// TIA Portal V17 program export: 3 tag tables, 14 data types, 19 data blocks, 63 code blocks (in call order from the OBs), 4 instance data blocks

VAR_GLOBAL   // PLC tag table "Default tag table"
   System_Byte AT %MB0 : Byte;
   FirstScan AT %M0.0 : Bool;
   DiagStatusUpdate AT %M0.1 : Bool;
   AlwaysTRUE AT %M0.2 : Bool;
   AlwaysFALSE AT %M0.3 : Bool;
   Clock_Byte AT %MB1 : Byte;
   Clock_10Hz AT %M1.0 : Bool;
   Clock_5Hz AT %M1.1 : Bool;
   "Clock_2.5Hz" AT %M1.2 : Bool;
   Clock_2Hz AT %M1.3 : Bool;
   "Clock_1.25Hz" AT %M1.4 : Bool;
   Clock_1Hz AT %M1.5 : Bool;
   "Clock_0.625Hz" AT %M1.6 : Bool;
   "Clock_0.5Hz" AT %M1.7 : Bool;
END_VAR

VAR_GLOBAL   // PLC tag table "CPG_Constants"
END_VAR
VAR_GLOBAL CONSTANT   // user constants
   CPG_NO_OF_ELEMENTS_EVENT_STATUS_UPPER_LIM : Int := 29;   // Number of Alarms, Warning and PackML Status events used by Event Status UDT (Array size of 0..x)
   CPG_NO_OF_ADMIN_EVENTS_UPPER_LIM : Int := 9;   // Number of Alarms and Warning events found in the PackTags Admin Area - active alarms / warnings. (Array size of 0..x)
   CPG_NO_OF_ADMIN_EVENTS_HISTORY_UPPER_LIM : Int := 9;   // Number of Alarms and Warning events found in the PackTags Admin Area - historical alarms / warnings. (Array size of 0..x)
   CPG_NO_OF_PROD_CONSUMED_COUNT_UPPER_LIM : Int := 0;   // Number of Prod Consumed Counter Array Size (PackTags Admin) (Array size of 0..x)
   CPG_NO_OF_PROD_PROCESSED_COUNT_UPPER_LIM : Int := 0;   // Number of Prod Processed Counter Array Size (PackTags Admin) (Array size of 0..x)
   CPG_NO_OF_PROD_DEFECTIVE_COUNT_UPPER_LIM : Int := 0;   // Number of Prod Defective Counter Array Size (PackTags Admin) (Array size of 0..x)
   CPG_NO_OF_STS_ELEMENTS_EVENT_SUM_UPPER_LIM : Int := 99;   // Number of Alarms, Warning and PackML Status events used by Event Summation UDT (Array size of 0..x)
   CPG_NO_OF_HMI_SORT_EVENTS_UPPER_LIM : Int := 19;   // Number of Alarms and Warning events found for the HMI area - sorted HMI alarms / warnings. (Array size of 0..x)
   CPG_NO_OF_CFG_ALARMS_UPPER_LIM : Int := 39;   // Number of Cfg Alarm event configurations (Array size of 0..x)
   CPG_NO_OF_CFG_WARNINGS_UPPER_LIM : Int := 29;   // Number of Cfg Warning event configurations (Array size of 0..x)
   CPG_NO_OF_CFG_STATUS_UPPER_LIM : Int := 19;   // Number of Cfg Status event configurations (Array size of 0..x)
   CPG_NO_OF_STATUS_PARAMETERS_UPPER_LIM : Int := 0;   // Number of Status Parameters (Array size of 0..x)
   CPG_NO_OF_COMMAND_PARAMETERS_UPPER_LIM : Int := 0;   // Number of Command Parameters (Array size of 0..x)
   CPG_NO_OF_ADMIN_PARAMETERS_UPPER_LIM : Int := 0;   // Number of Admin Parameters (Array size of 0..x)
   CPG_NO_OF_RECIPE_UPPER_LIM : Int := 20;   // Number of Project Recipies (Array size of 0..x)
   CPG_NO_OF_SETPOINT_REAL_UPPER_LIM : Int := 0;   // Number of Setpoints with a REAL type (Array size of 0..x)
   CPG_NO_OF_SETPOINT_DINT_UPPER_LIM : Int := 0;   // Number of Setpoints with a DINT type (Array size of 0..x)
   CPG_NO_OF_SETPOINT_BOOL_UPPER_LIM : Int := 0;   // Number of Setpoints with a BOOL type (Array size of 0..x)
   CPG_NO_OF_SETPOINT_STRING_UPPER_LIM : Int := 0;   // Number of Setpoints with a STRING type (Array size of 0..x)
   CPG_PARTEO_NO_OF_ERRORS_UPPER_LIM : Int := 100;   // Number of Unique Error IDs tracked by PARETO Error Blocks
END_VAR

VAR_GLOBAL   // PLC tag table "LPMLV30_Constants"
END_VAR
VAR_GLOBAL CONSTANT   // user constants
   LPMLV30_MODE_INVALID : DInt := 0;   // OMAC PackMLV30 unit mode Invalid
   LPMLV30_MODE_PRODUCTION : DInt := 1;   // OMAC PackMLV30 unit mode Production
   LPMLV30_MODE_MAINTENANCE : DInt := 2;   // OMAC PackMLV30 unit mode Maintenance
   LPMLV30_MODE_MANUAL : DInt := 3;   // OMAC PackMLV30 unit mode Manual
   LPMLV30_MODE_USER_01 : DInt := 4;   // OMAC PackMLV30 user-defined unit mode 01
   LPMLV30_MODE_USER_02 : DInt := 5;   // OMAC PackMLV30 user-defined unit mode 02
   LPMLV30_MODE_USER_03 : DInt := 6;   // OMAC PackMLV30 user-defined unit mode 03
   LPMLV30_MODE_USER_04 : DInt := 7;   // OMAC PackMLV30 user-defined unit mode 04
   LPMLV30_MODE_USER_05 : DInt := 8;   // OMAC PackMLV30 user-defined unit mode 05
   LPMLV30_MODE_USER_06 : DInt := 9;   // OMAC PackMLV30 user-defined unit mode 06
   LPMLV30_MODE_USER_07 : DInt := 10;   // OMAC PackMLV30 user-defined unit mode 07
   LPMLV30_MODE_USER_08 : DInt := 11;   // OMAC PackMLV30 user-defined unit mode 08
   LPMLV30_MODE_USER_09 : DInt := 12;   // OMAC PackMLV30 user-defined unit mode 09
   LPMLV30_MODE_USER_10 : DInt := 13;   // OMAC PackMLV30 user-defined unit mode 10
   LPMLV30_MODE_USER_11 : DInt := 14;   // OMAC PackMLV30 user-defined unit mode 11
   LPMLV30_MODE_USER_12 : DInt := 15;   // OMAC PackMLV30 user-defined unit mode 12
   LPMLV30_MODE_USER_13 : DInt := 16;   // OMAC PackMLV30 user-defined unit mode 13
   LPMLV30_MODE_USER_14 : DInt := 17;   // OMAC PackMLV30 user-defined unit mode 14
   LPMLV30_MODE_USER_15 : DInt := 18;   // OMAC PackMLV30 user-defined unit mode 15
   LPMLV30_MODE_USER_16 : DInt := 19;   // OMAC PackMLV30 user-defined unit mode 16
   LPMLV30_MODE_USER_17 : DInt := 20;   // OMAC PackMLV30 user-defined unit mode 17
   LPMLV30_MODE_USER_18 : DInt := 21;   // OMAC PackMLV30 user-defined unit mode 18
   LPMLV30_MODE_USER_19 : DInt := 22;   // OMAC PackMLV30 user-defined unit mode 19
   LPMLV30_MODE_USER_20 : DInt := 23;   // OMAC PackMLV30 user-defined unit mode 20
   LPMLV30_MODE_USER_21 : DInt := 24;   // OMAC PackMLV30 user-defined unit mode 21
   LPMLV30_MODE_USER_22 : DInt := 25;   // OMAC PackMLV30 user-defined unit mode 22
   LPMLV30_MODE_USER_23 : DInt := 26;   // OMAC PackMLV30 user-defined unit mode 23
   LPMLV30_MODE_USER_24 : DInt := 27;   // OMAC PackMLV30 user-defined unit mode 24
   LPMLV30_MODE_USER_25 : DInt := 28;   // OMAC PackMLV30 user-defined unit mode 25
   LPMLV30_MODE_USER_26 : DInt := 29;   // OMAC PackMLV30 user-defined unit mode 26
   LPMLV30_MODE_USER_27 : DInt := 30;   // OMAC PackMLV30 user-defined unit mode 27
   LPMLV30_MODE_USER_28 : DInt := 31;   // OMAC PackMLV30 user-defined unit mode 28
   LPMLV30_STATE_UNDEFINED : DInt := 0;   // OMAC PackMLV30 state Undefined
   LPMLV30_STATE_CLEARING : DInt := 1;   // OMAC PackMLV30 state Clearing
   LPMLV30_STATE_STOPPED : DInt := 2;   // OMAC PackMLV30 state Stopped
   LPMLV30_STATE_STARTING : DInt := 3;   // OMAC PackMLV30 state Starting
   LPMLV30_STATE_IDLE : DInt := 4;   // OMAC PackMLV30 state Idle
   LPMLV30_STATE_SUSPENDED : DInt := 5;   // OMAC PackMLV30 state Suspended
   LPMLV30_STATE_EXECUTE : DInt := 6;   // OMAC PackMLV30 state Execute
   LPMLV30_STATE_STOPPING : DInt := 7;   // OMAC PackMLV30 state Stopping
   LPMLV30_STATE_ABORTING : DInt := 8;   // OMAC PackMLV30 state Aborting
   LPMLV30_STATE_ABORTED : DInt := 9;   // OMAC PackMLV30 state Aborted
   LPMLV30_STATE_HOLDING : DInt := 10;   // OMAC PackMLV30 state Holding
   LPMLV30_STATE_HELD : DInt := 11;   // OMAC PackMLV30 state Held
   LPMLV30_STATE_UNHOLDING : DInt := 12;   // OMAC PackMLV30 state Unholding
   LPMLV30_STATE_SUSPENDING : DInt := 13;   // OMAC PackMLV30 state Suspending
   LPMLV30_STATE_UNSUSPENDING : DInt := 14;   // OMAC PackMLV30 state Unsuspending
   LPMLV30_STATE_RESETTING : DInt := 15;   // OMAC PackMLV30 state Resetting
   LPMLV30_STATE_COMPLETING : DInt := 16;   // OMAC PackMLV30 state Completing
   LPMLV30_STATE_COMPLETE : DInt := 17;   // OMAC PackMLV30 state Complete
   LPMLV30_CMD_UNDEFINED : DInt := 0;   // OMAC PackMLV30 control command Undefined
   LPMLV30_CMD_RESET : DInt := 1;   // OMAC PackMLV30 control command Reset
   LPMLV30_CMD_START : DInt := 2;   // OMAC PackMLV30 control command Start
   LPMLV30_CMD_STOP : DInt := 3;   // OMAC PackMLV30 control command Stop
   LPMLV30_CMD_HOLD : DInt := 4;   // OMAC PackMLV30 control command Hold
   LPMLV30_CMD_UNHOLD : DInt := 5;   // OMAC PackMLV30 control command Unhold
   LPMLV30_CMD_SUSPEND : DInt := 6;   // OMAC PackMLV30 control command Suspend
   LPMLV30_CMD_UNSUSPEND : DInt := 7;   // OMAC PackMLV30 control command Unsuspend
   LPMLV30_CMD_ABORT : DInt := 8;   // OMAC PackMLV30 control command Abort
   LPMLV30_CMD_CLEAR : DInt := 9;   // OMAC PackMLV30 control command Clear
   LPMLV30_CMD_COMPLETE : DInt := 10;   // OMAC PackMLV30 control command Complete
   LPMLV30_LANGUAGE_1 : Int := 0;   // Texts in 1st language (default English)
   LPMLV30_LANGUAGE_2 : Int := 1;   // Texts in 2nd language (default German)
   LPMLV30_DIAG_BUFFER_UPPER_LIM : Int := 15;   // Diagnostics buffer array upper boundary (0-based)
   LPMLV30_LANGUAGES_UPPER_LIM : Int := 2;   // (Number of languages - 1) -> Array[0..LPMLV30_LANGUAGES_UPPER_LIM]
   LPMLV30_MODES_UPPER_LIM : Int := 4;   // (Number of unit modes - 1) -> Array[0..LPMLV30_MODES_UPPER_LIM]
   LPMLV30_STATES_UPPER_LIM : Int := 17;   // (Number of states - 1) -> Array[0..LPMLV30_STATES_UPPER_LIM] (SHOULD ALWAYS BE 17!)
   LPMLV30_MAX_MODES_UPPER_LIM : Int := 31;   // (Maximum number of unit modes - 1) -> Array[0..LPMLV30_MAX_MODES_UPPER_LIM]
END_VAR

TYPE "CPG_typeEventCfg"
// stored: IsFailsafeCompliant false
   STRUCT
      ID : Int;   // ID Value - from PackTags Reason Code, 1=E-Stop pushed, 3=Main off, etc.
      value : Int;   // Reason Code 'Value' - allows for detailed breakdown of ID, ie 1=Discharge,
      message : Array[0.."LPMLV30_LANGUAGES_UPPER_LIM"] of String[60];   // Alarm Message - 0=English, 1=German, 2=Spanish, 3=Italian, 4=French
      category : Int;   // Category Value (0-9)
   END_STRUCT;
END_TYPE

TYPE "CPG_typeEventStatus"
// stored: IsFailsafeCompliant false
   STRUCT
      sts_FirstOutEvent { S7_SetPoint := 'True'} : "CPG_typeEvent";   // Event Info of the very first active event (irregardeless of the cat)
      sts_FirstOutEventCat { S7_SetPoint := 'True'} : Array[0..9] of "CPG_typeEvent";
      sts_Events { S7_SetPoint := 'True'} : Array[0.."CPG_NO_OF_ELEMENTS_EVENT_STATUS_UPPER_LIM"] of "CPG_typeEvent";
      sts_NumEvents : Int;   // Number of all current active events
      sts_NumAllEvents : Int;   // Number of all current events
      out_ZeroEvent { S7_SetPoint := 'True'} : "CPG_typeEvent";   // null event information
      sts_Category_0_Latched : Bool;   // Category 0 Event - latched (require reset cmd)
      sts_Category_1_Latched : Bool;   // Category 1 Event - latched (require reset cmd)
      sts_Category_2_Latched : Bool;   // Category 2 Event - latched (require reset cmd)
      sts_Category_3_Latched : Bool;   // Category 3 Event - latched (require reset cmd)
      sts_Category_4_Latched : Bool;   // Category 4 Event - latched (require reset cmd)
      sts_Category_5_Latched : Bool;   // Category 5 Event - latched (require reset cmd)
      sts_Category_6_Latched : Bool;   // Category 6 Event - latched (require reset cmd)
      sts_Category_7_Latched : Bool;   // Category 7 Event - latched (require reset cmd)
      sts_Category_8_Latched : Bool;   // Category 8 Event - latched (require reset cmd)
      sts_Category_9_Latched : Bool;   // Category 9 Event - latched (require reset cmd)
      sts_Category_0_NotLatched : Bool;   // Category 0 Event - NotLatched (currently active)
      sts_Category_1_NotLatched : Bool;   // Category 1 Event - NotLatched (currently active)
      sts_Category_2_NotLatched : Bool;   // Category 2 Event - NotLatched (currently active)
      sts_Category_3_NotLatched : Bool;   // Category 3 Event - NotLatched (currently active)
      sts_Category_4_NotLatched : Bool;   // Category 4 Event - NotLatched (currently active)
      sts_Category_5_NotLatched : Bool;   // Category 5 Event - NotLatched (currently active)
      sts_Category_6_NotLatched : Bool;   // Category 6 Event - NotLatched (currently active)
      sts_Category_7_NotLatched : Bool;   // Category 7 Event - NotLatched (currently active)
      sts_Category_8_NotLatched : Bool;   // Category 8 Event - NotLatched (currently active)
      sts_Category_9_NotLatched : Bool;   // Category 9 Event - NotLatched (currently active)
      sts_CurrentActiveEvent : Bool;   // Active # of Event
      wrk_ResetID : Int;   // Working Variable - DO NOT MODIFY
      wrk_EventArraySize : Int;   // Working Variable - DO NOT MODIFY
      wrk_UpdateEventListID : Int;   // Working Variable - DO NOT MODIFY
      wrk_LanguageSelection : Int;   // This is the value of language selected in the HMI
      wrk_MessagePrefix : String[10];   // Working Variable - DO NOT MODIFY
   END_STRUCT;
END_TYPE

TYPE "CPG_typeEventSummation"
// stored: IsFailsafeCompliant false
   STRUCT
      sts_FirstOutEvent { S7_SetPoint := 'True'} : "CPG_typeEvent";   // First Out (Stop Reason) Event
      sts_FirstOutEventCat { S7_SetPoint := 'True'} : Array[0..9] of "CPG_typeEvent";   // First Out (Stop Reason) Event by Category\
      sts_Events { S7_SetPoint := 'True'} : Array[0.."CPG_NO_OF_STS_ELEMENTS_EVENT_SUM_UPPER_LIM"] of "CPG_typeEvent";   // All Active Events
      sts_NumEvents : Int;   // Number of Active Events
      sts_Category_0_Latched : Bool;   // Category 0 Event - latched (require reset cmd)
      sts_Category_1_Latched : Bool;   // Category 1 Event - latched (require reset cmd)
      sts_Category_2_Latched : Bool;   // Category 2 Event - latched (require reset cmd)
      sts_Category_3_Latched : Bool;   // Category 3 Event - latched (require reset cmd)
      sts_Category_4_Latched : Bool;   // Category 4 Event - latched (require reset cmd)
      sts_Category_5_Latched : Bool;   // Category 5 Event - latched (require reset cmd)
      sts_Category_6_Latched : Bool;   // Category 6 Event - latched (require reset cmd)
      sts_Category_7_Latched : Bool;   // Category 7 Event - latched (require reset cmd)
      sts_Category_8_Latched : Bool;   // Category 8 Event - latched (require reset cmd)
      sts_Category_9_Latched : Bool;   // Category 9 Event - latched (require reset cmd)
      sts_Category_0_NotLatched : Bool;   // Category 0 Event - NotLatched (currently active)
      sts_Category_1_NotLatched : Bool;   // Category 1 Event - NotLatched (currently active)
      sts_Category_2_NotLatched : Bool;   // Category 2 Event - NotLatched (currently active)
      sts_Category_3_NotLatched : Bool;   // Category 3 Event - NotLatched (currently active)
      sts_Category_4_NotLatched : Bool;   // Category 4 Event - NotLatched (currently active)
      sts_Category_5_NotLatched : Bool;   // Category 5 Event - NotLatched (currently active)
      sts_Category_6_NotLatched : Bool;   // Category 6 Event - NotLatched (currently active)
      sts_Category_7_NotLatched : Bool;   // Category 7 Event - NotLatched (currently active)
      sts_Category_8_NotLatched : Bool;   // Category 8 Event - NotLatched (currently active)
      sts_Category_9_NotLatched : Bool;   // Category 9 Event - NotLatched (currently active)
      sts_CurrentActiveEvent : Bool;   // Event Active = 1, not active = 0
      wrk_EventArraySize : Int;   // Maximum Array Size - DO NOT MODIFY
      wrk_Category_0_Latched : Bool;   // Working Variable - DO NOT MODIFY
      wrk_Category_1_Latched : Bool;   // Working Variable - DO NOT MODIFY
      wrk_Category_2_Latched : Bool;   // Working Variable - DO NOT MODIFY
      wrk_Category_3_Latched : Bool;   // Working Variable - DO NOT MODIFY
      wrk_Category_4_Latched : Bool;   // Working Variable - DO NOT MODIFY
      wrk_Category_5_Latched : Bool;   // Working Variable - DO NOT MODIFY
      wrk_Category_6_Latched : Bool;   // Working Variable - DO NOT MODIFY
      wrk_Category_7_Latched : Bool;   // Working Variable - DO NOT MODIFY
      wrk_Category_8_Latched : Bool;   // Working Variable - DO NOT MODIFY
      wrk_Category_9_Latched : Bool;   // Working Variable - DO NOT MODIFY
      wrk_Category_0_NotLatched : Bool;   // Working Variable - DO NOT MODIFY
      wrk_Category_1_NotLatched : Bool;   // Working Variable - DO NOT MODIFY
      wrk_Category_2_NotLatched : Bool;   // Working Variable - DO NOT MODIFY
      wrk_Category_3_NotLatched : Bool;   // Working Variable - DO NOT MODIFY
      wrk_Category_4_NotLatched : Bool;   // Working Variable - DO NOT MODIFY
      wrk_Category_5_NotLatched : Bool;   // Working Variable - DO NOT MODIFY
      wrk_Category_6_NotLatched : Bool;   // Working Variable - DO NOT MODIFY
      wrk_Category_7_NotLatched : Bool;   // Working Variable - DO NOT MODIFY
      wrk_Category_8_NotLatched : Bool;   // Working Variable - DO NOT MODIFY
      wrk_Category_9_NotLatched : Bool;   // Working Variable - DO NOT MODIFY
      wrk_CurrentActiveEvent : Bool;   // Working Variable - DO NOT MODIFY
   END_STRUCT;
END_TYPE

TYPE "CPG_typeMessagePrefix"
// stored: IsFailsafeCompliant false
   STRUCT
      messagePrefix : Array[0.."LPMLV30_LANGUAGES_UPPER_LIM"] of String[30];   // Multi-Lingual Message for Prefix (i.e 0=EN, 1=DE, 2=SP/ES, 3=IT, 4=FR)
   END_STRUCT;
END_TYPE

TYPE "CPG_typePackML_ModuleSts"
// stored: IsFailsafeCompliant false
   STRUCT
      cmd_Reset : Bool;   // Reset
      sts_Resetting_SC : Bool;   // Resetting State Complete
      cmd_Start : Bool;   // Start
      sts_Starting_SC : Bool;   // Starting State Complete
      cmd_Stop : Bool;   // Stop
      sts_Stopping_SC : Bool;   // Stopping State Complete
      cmd_Hold : Bool;   // Hold
      sts_Holding_SC : Bool;   // Holding State Complete
      cmd_UnHold : Bool;   // UnHold
      sts_UnHolding_SC : Bool;   // UnHolding State Complete
      cmd_Suspend : Bool;   // Suspend
      sts_Suspending_SC : Bool;   // Suspending State Complete
      cmd_UnSuspend : Bool;   // UnSuspend
      sts_UnSuspending_SC : Bool;   // UnSuspending State Complete
      cmd_Abort : Bool;   // Abort
      sts_Aborting_SC : Bool;   // Aborting State Complete
      cmd_Clear : Bool;   // Clear
      sts_Clearing_SC : Bool;   // Clearing State Complete
      sts_Execute_SC : Bool;   // Execute State Complete
      sts_Completing_SC : Bool;   // Completing State Complete
      moduleActive : Bool;   // Module Active Bit
      ONS : Bool;   // Internal One Shot Bit - Do not modify
   END_STRUCT;
END_TYPE

TYPE "CPG_typeParameter(DINT)"
// stored: IsFailsafeCompliant false
   STRUCT
      ID : DInt;   // Parameter ID - This is the arbitrary (user defined) ID value of the parameter
      "Name" : String[24];   // Parameter Name - The literal parameter name is used to describe the parameter number and its associated value (e.g. Glue Temp)
      Unit : String[5];   // Parameter Unit of Measure - The parameter unit is used to describe the unit of measure of the parameter and its associated value (e.g. DegF)
      Value : DInt;   // Parameter Value - This is the numeric or string value of the parameter (e.g. 100)
   END_STRUCT;
END_TYPE

TYPE "CPG_typeParameter(Real)"
// stored: IsFailsafeCompliant false
   STRUCT
      ID : DInt;   // Parameter ID - This is the arbitrary (user defined) ID value of the parameter
      "Name" : String[24];   // Parameter Name - The literal parameter name is used to describe the parameter number and its associated value (e.g. Glue Temp)
      Unit : String[5];   // Parameter Unit of Measure - The parameter unit is used to describe the unit of measure of the parameter and its associated value (e.g. DegF)
      Value : Real;   // Parameter Value - This is the numeric or string value of the parameter (e.g. 100.2)
   END_STRUCT;
END_TYPE

TYPE "CPG_typeParameter(String)"
// stored: IsFailsafeCompliant false
   STRUCT
      ID : DInt;   // Parameter ID - This is the arbitrary (user defined) ID value of the parameter
      "Name" : String[24];   // Parameter Name - The literal parameter name is used to describe the parameter number and its associated value (e.g. Glue Temp)
      Unit : String[5];   // Parameter Unit of Measure - The parameter unit is used to describe the unit of measure of the parameter and its associated value (e.g. DegF)
      Value : String[24];   // Parameter Value - This is the numeric or string value of the parameter (e.g. '6ES7518-4AP00-0AB0')
   END_STRUCT;
END_TYPE

TYPE "CPG_typeProdCount(DINT)"
// stored: IsFailsafeCompliant false
   STRUCT
      ID : DInt;   // Product ID - This is the arbitrary (user defined) ID value of the consumed production material
      "Name" : String[24];   // Descriptive name - The name is used to literally describe the material ID, and its associated material
      Unit : String[5];   // Unit of measure - The unit tag is used to describe the names associated with a specific material used by the machine
      Count : DInt;   // Value - The count value is used as a variable for displaying information about the amount of consumed
      AccCount : DInt;   // Value - The accumulative count value is used as a variable for displaying information about the total amount of consumed production material
   END_STRUCT;
END_TYPE

TYPE "CPG_typeSortFilter"
// stored: IsFailsafeCompliant false
   STRUCT
      cmdFilterActiveEvents : Bool;   // Filter for Active events: 1=only show active events; 0=show all events
      cmdFilterCategory : Bool;   // Filter by Category: filter events to show only selected category number
      cmdSortCategory : Bool;   // Sort by Category: 1=sort events by ascending category number
      cfgTimeSortDirection : Bool;   // Sort by Time: 1=newest first; 0=oldest first
      cfgEventListOffset : Int;   // Commanded event list offset (used for scrolling)
      cfgFilterCategory : Int;   // Filter by Category: filtered category number
   END_STRUCT;
END_TYPE

TYPE "typeLPMLV30_Configuration"
TITLE = typeLPMLV30_Configuration
// Support: tech.team.motioncontrol@siemens.com 
// Fax: +49 (0) 9131/98-1297
// stored: IsFailsafeCompliant false
   STRUCT
      disabledUnitModes : Array[0.."LPMLV30_MAX_MODES_UPPER_LIM"] of Bool;   // TRUE: Disable unit mode xx
      disabledStatesInUnitModes : Array[0.."LPMLV30_MAX_MODES_UPPER_LIM"] of DInt;   // TRUE: Disable states in unit mode (bit number = state number)
   END_STRUCT;
   // disabledUnitModes[0..11] := false;
   // disabledUnitModes[12..31] := true;
   // disabledStatesInUnitModes[0..31] := 0;
END_TYPE

TYPE "typeLPMLV30_Diagnostics"
TITLE = typeLPMLV30_Diagnostics
// Support: tech.team.motioncontrol@siemens.com 
// Fax: +49 (0) 9131/98-1297
// stored: IsFailsafeCompliant false
   STRUCT
      bufferIndex : Int := -1;   // Index of actual buffer entry
      buffer { S7_SetPoint := 'True'} : Array[0.."LPMLV30_DIAG_BUFFER_UPPER_LIM"] of "typeLPMLV30_DiagnosticsEntry";   // Diagnostics information buffer
   END_STRUCT;
END_TYPE

TYPE "typeLPMLV30_DiagnosticsEntry"
TITLE = typeLPMLV30_DiagnosticsEntry
// Support: tech.team.motioncontrol@siemens.com 
// Fax: +49 (0) 9131/98-1297
// stored: IsFailsafeCompliant false
   STRUCT
      timestamp : DTL := DTL#1970-01-01-00:00:00;   // Timestamp for this entry
      UnitModeCurrent : Byte := 16#00;   // Current unit mode
      StateCurrent : Byte := 16#00;   // Current state
      UnitMode : Byte := 16#00;   // Requested unit mode
      CntrlCmd : Byte := 16#00;   // Request control command
      SC : Bool := false;   // State complete signal
      message : Byte := 16#00;   // Message for this entry
   END_STRUCT;
END_TYPE

TYPE "typeLPMLV30_NamesConfiguration"
TITLE = typeLPMLV30_NamesConfiguration
// Support: tech.team.motioncontrol@siemens.com 
// Fax: +49 (0) 9131/98-1297
// stored: IsFailsafeCompliant false
   STRUCT
      unitModesNames : Array[0.."LPMLV30_LANGUAGES_UPPER_LIM", 0.."LPMLV30_MODES_UPPER_LIM"] of String[18];   // Names of unit modes [First index language, Second unit mode no]
      statesNames : Array[0.."LPMLV30_LANGUAGES_UPPER_LIM", 0.."LPMLV30_STATES_UPPER_LIM"] of String[16];   // Names of states [First index language, Second state no]
   END_STRUCT;
   // unitModesNames[0,0] := 'Invalid';
   // unitModesNames[0,1] := 'Production';
   // unitModesNames[0,2] := 'Maintenance';
   // unitModesNames[0,3] := 'Manual';
   // unitModesNames[0,4] := 'User Mode 01';
   // unitModesNames[1,0] := 'Undefiniert';
   // unitModesNames[1,1] := 'Produktion';
   // unitModesNames[1,2] := 'Wartung';
   // unitModesNames[1,3] := 'Hand';
   // unitModesNames[1,4] := 'Benutzer Mode 01';
   // statesNames[0,0] := 'Undefined';
   // statesNames[0,1] := 'Clearing';
   // statesNames[0,2] := 'Stopped';
   // statesNames[0,3] := 'Starting';
   // statesNames[0,4] := 'Idle';
   // statesNames[0,5] := 'Suspended';
   // statesNames[0,6] := 'Execute';
   // statesNames[0,7] := 'Stopping';
   // statesNames[0,8] := 'Aborting';
   // statesNames[0,9] := 'Aborted';
   // statesNames[0,10] := 'Holding';
   // statesNames[0,11] := 'Held';
   // statesNames[0,12] := 'UnHolding';
   // statesNames[0,13] := 'Suspending';
   // statesNames[0,14] := 'UnSuspending';
   // statesNames[0,15] := 'Resetting';
   // statesNames[0,16] := 'Completing';
   // statesNames[0,17] := 'Complete';
   // statesNames[1,0] := 'Undefiniert';
   // statesNames[1,1] := 'Clearing';
   // statesNames[1,2] := 'Stopped';
   // statesNames[1,3] := 'Starting';
   // statesNames[1,4] := 'Idle';
   // statesNames[1,5] := 'Suspended';
   // statesNames[1,6] := 'Execute';
   // statesNames[1,7] := 'Stopping';
   // statesNames[1,8] := 'Aborting';
   // statesNames[1,9] := 'Aborted';
   // statesNames[1,10] := 'Holding';
   // statesNames[1,11] := 'Held';
   // statesNames[1,12] := 'UnHolding';
   // statesNames[1,13] := 'Suspending';
   // statesNames[1,14] := 'UnSuspending';
   // statesNames[1,15] := 'Resetting';
   // statesNames[1,16] := 'Completing';
   // statesNames[1,17] := 'Complete';
END_TYPE

DATA_BLOCK "EM00"   // DB31649
TITLE = EM00
{ S7_Optimized_Access := 'TRUE' }
AUTHOR : tech.team.motioncontrol@siemens.com
FAMILY : CPG
VERSION : 1.1
// Support: tech.team.motioncontrol@siemens.com
// stored: AutoNumber true, DBAccessibleFromOPCUA true, DBAccessibleFromWebserver true, IsOnlyStoredInLoadMemory false, IsRetainMemResEnabled false, IsWriteProtectedInAS false, MemoryReserve 100
   VAR
      PackML_Sts { ExternalWritable := 'False'} : Struct   // PackML Module Status - EM and all control modules
         Unit { ExternalWritable := 'False'; S7_SetPoint := 'True'} : "CPG_typePackML_ModuleSts";   // PackML Module Status - EM - master status
         Alarm { ExternalWritable := 'False'; S7_SetPoint := 'True'} : "CPG_typePackML_ModuleSts";   // PackML Module Status - alarm status
         CM01 { ExternalWritable := 'False'; S7_SetPoint := 'True'} : "CPG_typePackML_ModuleSts";   // PackML Module Status - CM 01
         CM02 { ExternalWritable := 'False'; S7_SetPoint := 'True'} : "CPG_typePackML_ModuleSts";   // PackML Module Status - CM 02
         CM03 { ExternalWritable := 'False'; S7_SetPoint := 'True'} : "CPG_typePackML_ModuleSts";   // PackML Module Status - CM 03
         CM04 { ExternalWritable := 'False'; S7_SetPoint := 'True'} : "CPG_typePackML_ModuleSts";   // PackML Module Status - CM 04
         CM05 { ExternalWritable := 'False'; S7_SetPoint := 'True'} : "CPG_typePackML_ModuleSts";   // PackML Module Status - CM 05
         CM06 { ExternalWritable := 'False'; S7_SetPoint := 'True'} : "CPG_typePackML_ModuleSts";   // PackML Module Status - CM 06
         CM07 { ExternalWritable := 'False'; S7_SetPoint := 'True'} : "CPG_typePackML_ModuleSts";   // PackML Module Status - CM 07
         CM08 { ExternalWritable := 'False'; S7_SetPoint := 'True'} : "CPG_typePackML_ModuleSts";   // PackML Module Status - CM 08
         CM09 { ExternalWritable := 'False'; S7_SetPoint := 'True'} : "CPG_typePackML_ModuleSts";   // PackML Module Status - CM 09
         CM10 { ExternalWritable := 'False'; S7_SetPoint := 'True'} : "CPG_typePackML_ModuleSts";   // PackML Module Status - CM 10
      END_STRUCT;
      Alarm { ExternalAccessible := 'False'; ExternalVisible := 'False'; ExternalWritable := 'False'; S7_SetPoint := 'True'} : "CPG_typeEventStatus";   // Alarm Event Status - EM00 Status
      Warning { ExternalAccessible := 'False'; ExternalVisible := 'False'; ExternalWritable := 'False'; S7_SetPoint := 'True'} : "CPG_typeEventStatus";   // Warning Event Status - EM00 Status
      Status { ExternalAccessible := 'False'; ExternalVisible := 'False'; ExternalWritable := 'False'; S7_SetPoint := 'True'} : "CPG_typeEventStatus";   // Event Status - EM00 Status
   END_VAR
BEGIN
END_DATA_BLOCK

DATA_BLOCK "EM01"   // DB31669
TITLE = EM01
{ S7_Optimized_Access := 'TRUE' }
AUTHOR : tech.team.motioncontrol@siemens.com
FAMILY : CPG
VERSION : 1.0
// Support: tech.team.motioncontrol@siemens.com
// Fax: +49 (0) 9131/98-1297
// stored: AutoNumber true, DBAccessibleFromOPCUA true, DBAccessibleFromWebserver true, IsOnlyStoredInLoadMemory false, IsRetainMemResEnabled false, IsWriteProtectedInAS false, MemoryReserve 100
   VAR
      PackML_Sts { ExternalWritable := 'False'} : Struct   // PackML Module Status - EM and all control modules
         Unit { ExternalWritable := 'False'; S7_SetPoint := 'True'} : "CPG_typePackML_ModuleSts";   // PackML Module Status - EM - master status
         Alarm { ExternalWritable := 'False'; S7_SetPoint := 'True'} : "CPG_typePackML_ModuleSts";   // PackML Module Status - alarm status
         CM01 { ExternalWritable := 'False'; S7_SetPoint := 'True'} : "CPG_typePackML_ModuleSts";   // PackML Module Status - CM 01
         CM02 { ExternalWritable := 'False'; S7_SetPoint := 'True'} : "CPG_typePackML_ModuleSts";   // PackML Module Status - CM 02
         CM03 { ExternalWritable := 'False'; S7_SetPoint := 'True'} : "CPG_typePackML_ModuleSts";   // PackML Module Status - CM 03
         CM04 { ExternalWritable := 'False'; S7_SetPoint := 'True'} : "CPG_typePackML_ModuleSts";   // PackML Module Status - CM 04
         CM05 { ExternalWritable := 'False'; S7_SetPoint := 'True'} : "CPG_typePackML_ModuleSts";   // PackML Module Status - CM 05
         CM06 { ExternalWritable := 'False'; S7_SetPoint := 'True'} : "CPG_typePackML_ModuleSts";   // PackML Module Status - CM 06
         CM07 { ExternalWritable := 'False'; S7_SetPoint := 'True'} : "CPG_typePackML_ModuleSts";   // PackML Module Status - CM 07
         CM08 { ExternalWritable := 'False'; S7_SetPoint := 'True'} : "CPG_typePackML_ModuleSts";   // PackML Module Status - CM 08
         CM09 { ExternalWritable := 'False'; S7_SetPoint := 'True'} : "CPG_typePackML_ModuleSts";   // PackML Module Status - CM 09
         CM10 { ExternalWritable := 'False'; S7_SetPoint := 'True'} : "CPG_typePackML_ModuleSts";   // PackML Module Status - CM 10
      END_STRUCT;
      Alarm { ExternalAccessible := 'False'; ExternalVisible := 'False'; ExternalWritable := 'False'; S7_SetPoint := 'True'} : "CPG_typeEventStatus";   // Alarm Event Status - EM01 Status
      Warning { ExternalAccessible := 'False'; ExternalVisible := 'False'; ExternalWritable := 'False'; S7_SetPoint := 'True'} : "CPG_typeEventStatus";   // Warning Event Status - EM01 Status
      Status { ExternalAccessible := 'False'; ExternalVisible := 'False'; ExternalWritable := 'False'; S7_SetPoint := 'True'} : "CPG_typeEventStatus";   // Event Status - EM01 Status
   END_VAR
BEGIN
END_DATA_BLOCK

DATA_BLOCK "EM02"   // DB31689
TITLE = EM02
{ S7_Optimized_Access := 'TRUE' }
AUTHOR : tech.team.motioncontrol@siemens.com
FAMILY : CPG
VERSION : 1.0
// Support: tech.team.motioncontrol@siemens.com
// Fax: +49 (0) 9131/98-1297
// stored: AutoNumber true, DBAccessibleFromOPCUA true, DBAccessibleFromWebserver true, IsOnlyStoredInLoadMemory false, IsRetainMemResEnabled false, IsWriteProtectedInAS false, MemoryReserve 100
   VAR
      PackML_Sts { ExternalWritable := 'False'} : Struct   // PackML Module Status - EM and all control modules
         Unit { ExternalWritable := 'False'; S7_SetPoint := 'True'} : "CPG_typePackML_ModuleSts";   // PackML Module Status - EM - master status
         Alarm { ExternalWritable := 'False'; S7_SetPoint := 'True'} : "CPG_typePackML_ModuleSts";   // PackML Module Status - alarm status
         CM01 { ExternalWritable := 'False'; S7_SetPoint := 'True'} : "CPG_typePackML_ModuleSts";   // PackML Module Status - CM 01
         CM02 { ExternalWritable := 'False'; S7_SetPoint := 'True'} : "CPG_typePackML_ModuleSts";   // PackML Module Status - CM 02
         CM03 { ExternalWritable := 'False'; S7_SetPoint := 'True'} : "CPG_typePackML_ModuleSts";   // PackML Module Status - CM 03
         CM04 { ExternalWritable := 'False'; S7_SetPoint := 'True'} : "CPG_typePackML_ModuleSts";   // PackML Module Status - CM 04
         CM05 { ExternalWritable := 'False'; S7_SetPoint := 'True'} : "CPG_typePackML_ModuleSts";   // PackML Module Status - CM 05
         CM06 { ExternalWritable := 'False'; S7_SetPoint := 'True'} : "CPG_typePackML_ModuleSts";   // PackML Module Status - CM 06
         CM07 { ExternalWritable := 'False'; S7_SetPoint := 'True'} : "CPG_typePackML_ModuleSts";   // PackML Module Status - CM 07
         CM08 { ExternalWritable := 'False'; S7_SetPoint := 'True'} : "CPG_typePackML_ModuleSts";   // PackML Module Status - CM 08
         CM09 { ExternalWritable := 'False'; S7_SetPoint := 'True'} : "CPG_typePackML_ModuleSts";   // PackML Module Status - CM 09
         CM10 { ExternalWritable := 'False'; S7_SetPoint := 'True'} : "CPG_typePackML_ModuleSts";   // PackML Module Status - CM 10
      END_STRUCT;
      Alarm { ExternalAccessible := 'False'; ExternalVisible := 'False'; ExternalWritable := 'False'; S7_SetPoint := 'True'} : "CPG_typeEventStatus";   // Alarm Event Status - EM02 Status
      Warning { ExternalAccessible := 'False'; ExternalVisible := 'False'; ExternalWritable := 'False'; S7_SetPoint := 'True'} : "CPG_typeEventStatus";   // Warning Event Status - EM02 Status
      Status { ExternalAccessible := 'False'; ExternalVisible := 'False'; ExternalWritable := 'False'; S7_SetPoint := 'True'} : "CPG_typeEventStatus";   // Event Status - EM02 Status
   END_VAR
BEGIN
END_DATA_BLOCK

DATA_BLOCK "Alarm"   // DB31610
TITLE = CPG_Alarm
{ S7_Optimized_Access := 'TRUE' }
AUTHOR : tech.team.motioncontrol@siemens.com
FAMILY : CPG
VERSION : 1.0
// Support: tech.team.motioncontrol@siemens.com
// Fax: +49 (0) 9131/98-1297
// stored: AutoNumber true, DBAccessibleFromOPCUA true, DBAccessibleFromWebserver true, IsOnlyStoredInLoadMemory false, IsRetainMemResEnabled false, IsWriteProtectedInAS false, MemoryReserve 0
   VAR
      Summation { ExternalWritable := 'False'; S7_SetPoint := 'True'} : "CPG_typeEventSummation";   // Unit Mode - Event Summation
   END_VAR
BEGIN
   Summation.wrk_EventArraySize := 30;
END_DATA_BLOCK

DATA_BLOCK "HMI_Data"   // DB31615
TITLE = CPG_HMI_Data
{ S7_Optimized_Access := 'TRUE' }
AUTHOR : tech.team.motioncontrol@siemens.com
FAMILY : CPG
VERSION : 1.0
// Support: tech.team.motioncontrol@siemens.com
// Fax: +49 (0) 9131/98-1297
// stored: AutoNumber true, DBAccessibleFromOPCUA true, DBAccessibleFromWebserver true, IsOnlyStoredInLoadMemory false, IsRetainMemResEnabled false, IsWriteProtectedInAS false, MemoryReserve 0
   VAR
      resetPackMLTimers : Bool;   // Reset the PackML Timer values when set (1).
   END_VAR
   VAR RETAIN
      languageSelected : Int;   // This is the value of the language selected in the HMI (0=English, 1=DE, 2=SP, 3
   END_VAR
   VAR
      modeCurrentTime { ExternalWritable := 'False'} : DInt;   // Time spent in the current mode [seconds](reset each time new mode is entered)
      modeCumulativeTime { ExternalWritable := 'False'} : DInt;   // Accumulative Time spent in the current mode [seconds]
      State_Current_Times { ExternalWritable := 'False'} : Array[0.."LPMLV30_STATES_UPPER_LIM"] of DInt;   // Current Time (# of seconds) spent for each state for active mode.
      State_Cumulative_Times { ExternalWritable := 'False'} : Array[0.."LPMLV30_STATES_UPPER_LIM"] of DInt;   // Accumulative Time (# of seconds) spent for each state for active mode.
      alarmSortedList { ExternalWritable := 'False'; S7_SetPoint := 'True'} : Array[0.."CPG_NO_OF_HMI_SORT_EVENTS_UPPER_LIM"] of "CPG_typeEvent";   // Alarm Sorted List for HMI - summary of Active Events
      EM_SortDisable_Alarm : Struct   // Alarm Disable for Equipment Modules (EMs)
         Unit : Bool;   // If bool is reset, then Unit sort filter is enabled, else it's disabled.
         EM00 : Bool;   // If bool is reset, then EMxx sort filter is enabled, else it's disabled.
         EM01 : Bool;   // If bool is reset, then EMxx sort filter is enabled, else it's disabled.
         EM02 : Bool;   // If bool is reset, then EMxx sort filter is enabled, else it's disabled.
         EM03 : Bool;   // If bool is reset, then EMxx sort filter is enabled, else it's disabled.
         EM04 : Bool;   // If bool is reset, then EMxx sort filter is enabled, else it's disabled.
         EM05 : Bool;   // If bool is reset, then EMxx sort filter is enabled, else it's disabled.
         EM06 : Bool;   // If bool is reset, then EMxx sort filter is enabled, else it's disabled.
         EM07 : Bool;   // If bool is reset, then EMxx sort filter is enabled, else it's disabled.
         EM08 : Bool;   // If bool is reset, then EMxx sort filter is enabled, else it's disabled.
         EM09 : Bool;   // If bool is reset, then EMxx sort filter is enabled, else it's disabled.
         EM10 : Bool;   // If bool is reset, then EMxx sort filter is enabled, else it's disabled.
      END_STRUCT;
      alarmFilter { S7_SetPoint := 'True'} : "CPG_typeSortFilter";   // HMI Commands to control the Alarm Sort Filter
      warningSortedList { ExternalWritable := 'False'; S7_SetPoint := 'True'} : Array[0.."CPG_NO_OF_HMI_SORT_EVENTS_UPPER_LIM"] of "CPG_typeEvent";   // Warning Sorted List for HMI - summary of Active Events
      EMSortDisableWarning : Struct   // Warning Disable for Equipment Modules (EMs)
         Unit : Bool;   // If bool is reset, then Unit sort filter is enabled, else it's disabled.
         EM00 : Bool;   // If bool is reset, then EMxx sort filter is enabled, else it's disabled.
         EM01 : Bool;   // If bool is reset, then EMxx sort filter is enabled, else it's disabled.
         EM02 : Bool;   // If bool is reset, then EMxx sort filter is enabled, else it's disabled.
         EM03 : Bool;   // If bool is reset, then EMxx sort filter is enabled, else it's disabled.
         EM04 : Bool;   // If bool is reset, then EMxx sort filter is enabled, else it's disabled.
         EM05 : Bool;   // If bool is reset, then EMxx sort filter is enabled, else it's disabled.
         EM06 : Bool;   // If bool is reset, then EMxx sort filter is enabled, else it's disabled.
         EM07 : Bool;   // If bool is reset, then EMxx sort filter is enabled, else it's disabled.
         EM08 : Bool;   // If bool is reset, then EMxx sort filter is enabled, else it's disabled.
         EM09 : Bool;   // If bool is reset, then EMxx sort filter is enabled, else it's disabled.
         EM10 : Bool;   // If bool is reset, then EMxx sort filter is enabled, else it's disabled.
      END_STRUCT;
      WarningFilter { S7_SetPoint := 'True'} : "CPG_typeSortFilter";   // HMI Commands to control the Warning Sort Filter
      HMIWarningMsgScroll { ExternalWritable := 'False'} : String[40];   // Warning Message - scroll of all active warnings
      ModeNames { ExternalWritable := 'False'} : Array[0.."LPMLV30_MODES_UPPER_LIM"] of String[18];   // Mode Names for selected language
      StateNames { ExternalWritable := 'False'} : Array[0.."LPMLV30_STATES_UPPER_LIM"] of String[16];   // State Names for selectecd modes
      PLCDateTime { ExternalWritable := 'False'} : Struct   // Date Time for WinCC Flexible HMI format
         DATE_TIME { ExternalWritable := 'False'} : Date_And_Time := DT#12-7-12-18:16:34.356;   // Current Time and Date of PLC
         reserve { ExternalWritable := 'False'} : Array[0..3] of Byte;   // Filler bytes used to sync HMI clock with PLC clock. Do not change.
      END_STRUCT;
      diagnosticsBufferIndexForHMI { ExternalWritable := 'False'} : Int;   // Diagnostics to HMI
      diagnosticsBufferEntryForHMI { ExternalWritable := 'False'; S7_SetPoint := 'True'} : "typeLPMLV30_DiagnosticsEntry";   // Diagnostics to HMI
      HMICoordination { ExternalWritable := 'False'} : Word;   // HMI Coordination area pointer: Bit0 = Startup; 1=OpMode (0=on, 1=off-line), 2=life bit
      HMICurrentScreenID : Int;   // HMI Current screen number
      CMDs : Struct   // HMI Commands
         PB_Start : Bool;   // HMI Push Button Command - Start
         PB_Stop : Bool;   // HMI Push Button Command - Stop
         PB_Hold : Bool;   // HMI Push Button Command - Hold
         PB_Reset : Bool;   // HMI Push Button Command - Reset
         PB_Complete : Bool;   // HMI Push Button Command - Complete (demo purposes only)
         PB_EStop : Bool;   // HMI Push Button Command - EStop (demo purposes only)
         PB_Abort : Bool;   // HMI Push Button Command - Abort (demo purposes only)
         PB_ProdSimulate : Bool;   // HMI Push Button Command - Product Simulate Enable (demo purposes only)
         PB_DriveSimulate : Bool;   // HMI Push Button Command - Drive / Axis Simulate (demo purposes only)
      END_STRUCT;
   END_VAR
BEGIN
END_DATA_BLOCK

DATA_BLOCK "HMI_Data_Custom"   // DB31616
TITLE = CPG_HMI_Data_Custom
{ S7_Optimized_Access := 'TRUE' }
AUTHOR : tech.team.motioncontrol@siemens.com
FAMILY : CPG
VERSION : 1.0
// Support: tech.team.motioncontrol@siemens.com
// Fax: +49 (0) 9131/98-1297
// stored: AutoNumber true, DBAccessibleFromOPCUA true, DBAccessibleFromWebserver true, IsOnlyStoredInLoadMemory false, IsRetainMemResEnabled false, IsWriteProtectedInAS false, MemoryReserve 0
   VAR
      machineSpeedSP : Real := 20.0;   // Machine Speed Setpoint (product per min)
      machineSpeedPV { ExternalWritable := 'False'} : Real;   // Machine Speed Actual (product per min)
   END_VAR
BEGIN
END_DATA_BLOCK

DATA_BLOCK "PackML"   // DB31613
TITLE = CPG_PackML
{ S7_Optimized_Access := 'TRUE' }
AUTHOR : tech.team.motioncontrol@siemens.com
FAMILY : CPG
VERSION : 1.0
// Support: tech.team.motioncontrol@siemens.com
// Fax: +49 (0) 9131/98-1297
// stored: AutoNumber true, DBAccessibleFromOPCUA true, DBAccessibleFromWebserver true, IsOnlyStoredInLoadMemory false, IsRetainMemResEnabled false, IsWriteProtectedInAS false, MemoryReserve 0
   VAR
      projectVersion { ExternalWritable := 'False'} : String[10] := 'V1.0.0';   // Project specific version
      Cmd : Struct   // PackML boolean COMMAND to PackML ModeManager & State Model
         Mode : Struct   // Boolean command to change the MODE
            Production : Bool;   // Request to goto mode - PRODUCTION (mode #1)
            Maintenance : Bool;   // Request to goto mode - MAINTENANCE (mode #2)
            Manual : Bool;   // Request to goto mode - MANUAL (mode #3)
            UserMode01 : Bool;   // Request to goto mode - USER MODE 01 (mode #4)
            UserMode02 : Bool;   // Request to goto mode - USER MODE 02 (mode #5)
            UserMode03 : Bool;   // Request to goto mode - USER MODE 03 (mode #6)
            UserMode04 : Bool;   // Request to goto mode - USER MODE 04 (mode #7)
            UserMode05 : Bool;   // Request to goto mode - USER MODE 05 (mode #8)
            UserMode06 : Bool;   // Request to goto mode - USER MODE 06 (mode #9)
            UserMode07 : Bool;   // Request to goto mode - USER MODE 07 (mode #10)
            UserMode08 : Bool;   // Request to goto mode - USER MODE 08 (mode #11)
         END_STRUCT;
      END_STRUCT;
      Sts { ExternalWritable := 'False'} : Struct   // Status for current mode and state as boolean
         Mode { ExternalWritable := 'False'} : Struct   // Status of the current MODE
            Production { ExternalWritable := 'False'} : Bool;   // Current mode - PRODUCTION (mode #1)
            Maintenance { ExternalWritable := 'False'} : Bool;   // Current mode - MAINTENANCE (mode #2)
            Manual { ExternalWritable := 'False'} : Bool;   // Current mode - MANUAL (mode #3)
            UserMode01 { ExternalWritable := 'False'} : Bool;   // Current mode - USER MODE 01 (mode #4)
            UserMode02 { ExternalWritable := 'False'} : Bool;   // Current mode - USER MODE 02 (mode #5)
            UserMode03 { ExternalWritable := 'False'} : Bool;   // Current mode - USER MODE 03 (mode #6)
            UserMode04 { ExternalWritable := 'False'} : Bool;   // Current mode - USER MODE 04 (mode #7)
            UserMode05 { ExternalWritable := 'False'} : Bool;   // Current mode - USER MODE 05 (mode #8)
            UserMode06 { ExternalWritable := 'False'} : Bool;   // Current mode - USER MODE 06 (mode #9)
            UserMode07 { ExternalWritable := 'False'} : Bool;   // Current mode - USER MODE 07 (mode #10)
            UserMode08 { ExternalWritable := 'False'} : Bool;   // Current mode - USER MODE 08 (mode #11)
         END_STRUCT;
         State { ExternalWritable := 'False'} : Struct   // Status of the current STATE
            Clearing { ExternalWritable := 'False'} : Bool;   // Current state is - Clearing
            Stopped { ExternalWritable := 'False'} : Bool;   // Current state is - Stopped
            Starting { ExternalWritable := 'False'} : Bool;   // Current state is - Starting
            Idle { ExternalWritable := 'False'} : Bool;   // Current state is - Idle
            Suspended { ExternalWritable := 'False'} : Bool;   // Current state is - Suspended
            Execute { ExternalWritable := 'False'} : Bool;   // Current state is - Executing
            Stopping { ExternalWritable := 'False'} : Bool;   // Current state is - Stopping
            Aborting { ExternalWritable := 'False'} : Bool;   // Current state is - Aborting
            Aborted { ExternalWritable := 'False'} : Bool;   // Current state is - Aborted
            Holding { ExternalWritable := 'False'} : Bool;   // Current state is - Holding
            Held { ExternalWritable := 'False'} : Bool;   // Current state is - Held
            Unholding { ExternalWritable := 'False'} : Bool;   // Current state is - Unholding
            Suspending { ExternalWritable := 'False'} : Bool;   // Current state is - Suspending
            Unsuspending { ExternalWritable := 'False'} : Bool;   // Current state is - Unsuspending
            Resetting { ExternalWritable := 'False'} : Bool;   // Current state is - Resetting
            Completing { ExternalWritable := 'False'} : Bool;   // Current state is - Completing
            Complete { ExternalWritable := 'False'} : Bool;   // Current state is - Complete
         END_STRUCT;
      END_STRUCT;
      Cmd_Reset : Bool;   // Request for command - RESET
      Cmd_Start : Bool;   // Request for command - START
      Cmd_Stop : Bool;   // Request for command - STOP
      Cmd_Hold : Bool;   // Request for command - HOLD
      Cmd_UnHold : Bool;   // Request for command - UNHOLD
      Cmd_Suspend : Bool;   // Request for command - SUSPEND
      Cmd_UnSuspend : Bool;   // Request for command - UNSUSPEND
      Cmd_Abort : Bool;   // Request for command - ABORT
      Cmd_Clear : Bool;   // Request for command - CLEAR
      Cmd_Complete : Bool;   // Request for command - COMPLETE
      remoteCommandEnable : Bool;   // If 0 = local mode for PackML commands, if 1=remote command for PackML
      OEE { ExternalWritable := 'False'} : Struct   // Real-Time OEE values
         realTime { ExternalWritable := 'False'} : Real;   // Real-Time value (0-100%)
         availability { ExternalWritable := 'False'} : Real;   // Availability value (0-100%)
         performance { ExternalWritable := 'False'} : Real;   // Performance value (0-100%)
         quality { ExternalWritable := 'False'} : Real;   // Quality value (0-100%)
      END_STRUCT;
      PackMLDiag { ExternalWritable := 'False'; S7_SetPoint := 'True'} : "typeLPMLV30_Diagnostics";   // PackML Diagnostic Data
   END_VAR
BEGIN
END_DATA_BLOCK

DATA_BLOCK "PackTags"   // DB31614
TITLE = CPG_PackTags
{ S7_Optimized_Access := 'TRUE' }
AUTHOR : tech.team.motioncontrol@siemens.com
FAMILY : CPG
VERSION : 1.0
// Support: tech.team.motioncontrol@siemens.com
// Fax: +49 (0) 9131/98-1297
// stored: AutoNumber true, DBAccessibleFromOPCUA true, DBAccessibleFromWebserver true, IsOnlyStoredInLoadMemory false, IsRetainMemResEnabled false, IsWriteProtectedInAS false, MemoryReserve 0
   VAR
      Command : Struct   // PackTags "Command" tag area. Data is scalable for needs.
         UnitMode : DInt;   // Unit Mode Target (1=Production,2=Maintenance,3=Manual,4=UserMode1,...,31=UserMode28)
         UnitModeChangeRequest : Bool;   // 1=Request Unit Mode Change to commanded value (UnitMode)
         MachSpeed : Real := 0.0;   // Setpoint of Machine Speed in Primary Packages per Minute
         MaterialInterlock : DWord;   // Materials Interlock Command (1=Ready or Not low, 0=Not ready or Low)
         CntrlCmd : DInt;   // State Control Command to drive a state change (1=Reset,2=Start,3=Stop,4=Hold,5=Unhold,6=Suspend,7=Unsuspend,8=Abort,9=Clear)
         CmdChangeRequest : Bool;   // 1=Request Machine State Change to commanded value (CntrlCmd)
         Parameter { S7_SetPoint := 'True'} : Array[0.."CPG_NO_OF_COMMAND_PARAMETERS_UPPER_LIM"] of "CPG_typeParameter(Real)";   // Parameter Structure Array from SCADA / MES
      END_STRUCT;
      Status { ExternalWritable := 'False'} : Struct   // PackTags "Status" tag area. Data is scalable for needs.
         UnitModeCurrent { ExternalWritable := 'False'} : DInt := 3;   // Current Unit Mode (1=Production,2=Maintenance,3=Manual,4=UserMode1,...,31=UserMode28)
         UnitModeCurrentName { ExternalWritable := 'False'} : String[18] := 'Manual';   // Current Unit Mode Name (NOT ISA-TR88 - OPTIONAL)
         UnitModeRequested { ExternalWritable := 'False'} : Bool;   // 1=Ack. that a unit mode change has been requested
         UnitModeChangeInProcess { ExternalWritable := 'False'} : Bool;   // 1=Requested Unit Mode Change In Progress
         StateCurrent { ExternalWritable := 'False'} : DInt := 2;   // Current Machine State (1=Clearing,2=Stopped,3=Starting,4=Idle,5=Suspended,6=Execute,7=Stopping,8=Aborting,9=Aborted,10=Holding,11=Held,12=Unholding,13=Suspending,14=Unsuspending,15=Resetting,16=Completing,17=Complete)
         StateCurrentName { ExternalWritable := 'False'} : String[16] := 'Stopped';   // Current Machine State name (NOT ISA-TR88 - OPTIONAL)
         StateRequested { ExternalWritable := 'False'} : DInt;   // Target Machine State
         StateChangeInProcess { ExternalWritable := 'False'} : Bool;   // 1=Requested State Change in Progress
         MachSpeed { ExternalWritable := 'False'} : Real := 0.0;   // Setpoint of Machine Speed in Primary Packages per Minute
         CurMachSpeed { ExternalWritable := 'False'} : Real := 0.0;   // Actual Value of Machine Speed in Primary Packages per Minute
         MaterialInterlock { ExternalWritable := 'False'} : DWord;   // Materials Interlock Status (1=Ready or Not low, 0=Not ready or Low)
         EquipmentInterlock { ExternalWritable := 'False'} : Struct   // Machine upstream and downstream status
            Blocked { ExternalWritable := 'False'} : Bool;   // 1=The downstream system is not able to accept products, 0=all OK
            Starved { ExternalWritable := 'False'} : Bool;   // 1=The upstream system is not able to supply products, 0=all OK
         END_STRUCT;
         Parameter { ExternalWritable := 'False'; S7_SetPoint := 'True'} : Array[0.."CPG_NO_OF_STATUS_PARAMETERS_UPPER_LIM"] of "CPG_typeParameter(Real)";   // Parameter Structure Array for HMI / SCADA / MES
      END_STRUCT;
   END_VAR
   VAR RETAIN
      Admin { ExternalWritable := 'False'} : Struct   // PackTags "Administration" tag area. Data is scalable for needs.
         Parameter { ExternalWritable := 'False'; S7_SetPoint := 'True'} : Array[0.."CPG_NO_OF_ADMIN_PARAMETERS_UPPER_LIM"] of "CPG_typeParameter(Real)";   // Parameter Structure Array for HMI / SCADA / MES
         Alarm { ExternalWritable := 'False'; S7_SetPoint := 'True'} : Array[0.."CPG_NO_OF_ADMIN_EVENTS_UPPER_LIM"] of "CPG_typeEvent";   // Alarm summary of Active Events
         AlarmExtent { ExternalWritable := 'False'} : DInt;   // Number of active alarms
         AlarmHistory { ExternalWritable := 'False'; S7_SetPoint := 'True'} : Array[0.."CPG_NO_OF_ADMIN_EVENTS_HISTORY_UPPER_LIM"] of "CPG_typeEvent";   // Alarm History
         AlarmHistoryExtent { ExternalWritable := 'False'} : DInt;   // Number of alarms in alarm history
         StopReason { ExternalWritable := 'False'; S7_SetPoint := 'True'} : "CPG_typeEvent";   // First Fault Alarm Code
         Warning { ExternalWritable := 'False'; S7_SetPoint := 'True'} : Array[0.."CPG_NO_OF_ADMIN_EVENTS_UPPER_LIM"] of "CPG_typeEvent";   // Active Machine Warnings
         WarningExtent { ExternalWritable := 'False'} : DInt;   // Number of Active Machine Warnings
         ModeCurrentTime { ExternalWritable := 'False'} : Array[0.."LPMLV30_MODES_UPPER_LIM"] of DInt;   // Time spent in the last mode [seconds] (reset each time new mode is entered)
         ModeCumulativeTime { ExternalWritable := 'False'} : Array[0.."LPMLV30_MODES_UPPER_LIM"] of DInt;   // Cumulative Time for all Modes [seconds]
         StateCurrentTime { ExternalWritable := 'False'} : Array[0.."LPMLV30_MODES_UPPER_LIM", 0.."LPMLV30_STATES_UPPER_LIM"] of DInt;   // Time spent in the last state [seconds] (reset each time new state is entered)
         StateCumulativeTime { ExternalWritable := 'False'} : Array[0.."LPMLV30_MODES_UPPER_LIM", 0.."LPMLV30_STATES_UPPER_LIM"] of DInt;   // Cumulative Time for all States [seconds]
         ProdConsumedCount { ExternalWritable := 'False'; S7_SetPoint := 'True'} : Array[0.."CPG_NO_OF_PROD_CONSUMED_COUNT_UPPER_LIM"] of "CPG_typeProdCount(DINT)";   // Total Number of Products consumed- good or bad
         ProdProcessedCount { ExternalWritable := 'False'; S7_SetPoint := 'True'} : Array[0.."CPG_NO_OF_PROD_PROCESSED_COUNT_UPPER_LIM"] of "CPG_typeProdCount(DINT)";   // Total Number of Products processed - good or bad
         ProdDefectiveCount { ExternalWritable := 'False'; S7_SetPoint := 'True'} : Array[0.."CPG_NO_OF_PROD_DEFECTIVE_COUNT_UPPER_LIM"] of "CPG_typeProdCount(DINT)";   // Total Number of Defective (bad) Products processed
         AccTimeSinceLastReset { ExternalWritable := 'False'} : DInt := L#0;   // Accumulated Time Since Last Reset of all mode and state times and counts
         MachDesignSpeed { ExternalWritable := 'False'} : Real := 0.0;   // Machine Design Speed of the Current Product Configuration
         StatesDisabled { ExternalWritable := 'False'} : DInt;   // States 1 to 17 of the PackML State Model can be disabled by turning on the corresponding bit in the DINT
         PLCDateTime { ExternalWritable := 'False'} : Array[0..6] of DInt;   // Current Date and Time of PLC
         PLCDateTimeDTL { ExternalWritable := 'False'} : DTL;   // Current Date and LTime (DTL) of PLC (date and time-of-day information in nanoseconds since 01/01/1970 0:0)
      END_STRUCT;
   END_VAR
BEGIN
   Admin.ProdConsumedCount[0]."Name" := 'Consumed #1';
   Admin.ProdConsumedCount[0].Unit := 'count';
   Admin.ProdProcessedCount[0]."Name" := 'Processed #1';
   Admin.ProdProcessedCount[0].Unit := 'count';
   Admin.ProdDefectiveCount[0]."Name" := 'Defective #1';
   Admin.ProdDefectiveCount[0].Unit := 'count';
END_DATA_BLOCK

DATA_BLOCK "ParetoData"   // DB31617
TITLE = CPG_ParetoData
{ S7_Optimized_Access := 'TRUE' }
AUTHOR : tech.team.motioncontrol@siemens.com
FAMILY : CPG
VERSION : 1.1
// Support: tech.team.motioncontrol@siemens.com
// stored: AutoNumber true, DBAccessibleFromOPCUA true, DBAccessibleFromWebserver true, IsOnlyStoredInLoadMemory false, IsRetainMemResEnabled false, IsWriteProtectedInAS false, MemoryReserve 0
   VAR RETAIN
      alarmOccurrence { S7_SetPoint := 'True'} : Array[0.."CPG_PARTEO_NO_OF_ERRORS_UPPER_LIM"] of "CPG_typePareto";   // Alarm Array
      totalStops : Int;   // Total stops on the machine
      totalTimeSinceReset : Real;   // Total time since reset
      totalUptime : Real;   // Total uptime of the machine
      totalDowntime : Real;   // Total downtime of the machine
      percentUptime : Real;
      MTTR : Real;
      MTBF : Real;
      Sort : Int;
      Reset : Bool;
   END_VAR
BEGIN
END_DATA_BLOCK

DATA_BLOCK "RecipeManagement"   // DB31618
TITLE = CPG_RecipeManagement
{ S7_Optimized_Access := 'TRUE' }
AUTHOR : tech.team.motioncontrol@siemens.com
FAMILY : CPG
VERSION : 1.1
// Support: tech.team.motioncontrol@siemens.com
// stored: AutoNumber true, DBAccessibleFromOPCUA true, DBAccessibleFromWebserver true, IsOnlyStoredInLoadMemory false, IsRetainMemResEnabled false, IsWriteProtectedInAS false, MemoryReserve 0
   VAR
      HMI_Command : Struct   // Helper bits for HMI Recipe Control
         Change : Struct
            changeCmd : Bool;
            changeID : Int;
            cancel : Bool;
            request : Bool;
         END_STRUCT;
         Save : Struct
            saveCmd : Bool;
            saveAsCmd : Bool;
            saveAsDestinationID : Int;
            saveAsNewName : String[60];
            cancel : Bool;
            request : Bool;
         END_STRUCT;
         Copy : Struct
            copyCmd : Bool;
            copySourceID : Int;
            copyDestinationID : Int;
            copyNewName : String[60];
            cancel : Bool;
            request : Bool;
         END_STRUCT;
         Delete : Struct
            deleteCmd : Bool;
            deleteID : Int;
            cancel : Bool;
            request : Bool;
         END_STRUCT;
         resetAllTimes : Bool;
      END_STRUCT;
      HMI_Indicator : Struct   // Helper bits for HMI Recipe Control
         changeConfirm : Bool;
         saveAsConfirm : Bool;
         copyConfirm : Bool;
         deleteConfirm : Bool;
         changeErr : Bool;
         saveAsErr : Bool;
         copyErr : Bool;
         deleteErr : Bool;
      END_STRUCT;
      setpointsArray_REAL { S7_SetPoint := 'True'} : Array[0..11] of "CPG_typeRecipeSetpoint_REAL";   // The setpoints that are displayed
      setpointsArray_DINT { S7_SetPoint := 'True'} : Array[0..11] of "CPG_typeRecipeSetpoint_DINT";   // The setpoints that are displayed
      setpointsArray_BOOL { S7_SetPoint := 'True'} : Array[0..11] of "CPG_typeRecipeSetpoint_BOOL";   // The setpoints that are displayed
      setpointsArray_STRING { S7_SetPoint := 'True'} : Array[0..11] of "CPG_typeRecipeSetpoint_STRING";   // The setpoints that are displayed
      setpointPopup_REAL { S7_SetPoint := 'True'} : "CPG_typeRecipeSetpoint_REAL";   // The setpoint in the popup
      setpointPopup_DINT { S7_SetPoint := 'True'} : "CPG_typeRecipeSetpoint_DINT";   // The setpoint in the popup
      setpointPopup_BOOL { S7_SetPoint := 'True'} : "CPG_typeRecipeSetpoint_BOOL";   // The setpoint in the popup
      setpointPopup_STRING { S7_SetPoint := 'True'} : "CPG_typeRecipeSetpoint_STRING";   // The setpoint in the popup
      popupTrackers : Array[0..3] of Int;   // Int to track the location of popup
      currentPages : Array[0..4] of Int;   // Current page of setpoints (or recipes)
      maxPages : Array[0..4] of Int;   // Max page of setpoints (or recipes)
      displayDisable_REAL : Array[0..11] of Bool;   // True if that setpoint should be hidden
      displayDisable_DINT : Array[0..11] of Bool;   // True if that setpoint should be hidden
      displayDisable_BOOL : Array[0..11] of Bool;   // True if that setpoint should be hidden
      displayDisable_STRING : Array[0..11] of Bool;   // True if that setpoint should be hidden
      recipeArrayNames : Array[0..19] of String[60];   // Recipe names to display
      recipeArraySaves : Array[0..19] of DTL;   // Recipe times to display
      recipeArrayTimes : Array[0..19] of Time;   // Recipe savepoints to display
      recipeArrayNums : Array[0..19] of Int;   // Recipe numbers
      recipeArrayHide : Array[0..19] of Bool;   // True if that recipe should be hidden
   END_VAR
BEGIN
   currentPages[0..4] := 1;
   maxPages[0..3] := 1;
END_DATA_BLOCK

DATA_BLOCK "Status"   // DB31612
TITLE = CPG_Status
{ S7_Optimized_Access := 'TRUE' }
AUTHOR : tech.team.motioncontrol@siemens.com
FAMILY : CPG
VERSION : 1.0
// Support: tech.team.motioncontrol@siemens.com
// Fax: +49 (0) 9131/98-1297
// stored: AutoNumber true, DBAccessibleFromOPCUA true, DBAccessibleFromWebserver true, IsOnlyStoredInLoadMemory false, IsRetainMemResEnabled false, IsWriteProtectedInAS false, MemoryReserve 0
   VAR
      Summation { ExternalWritable := 'False'; S7_SetPoint := 'True'} : "CPG_typeEventSummation";   // Unit Mode - PackML Event Summation
   END_VAR
BEGIN
   Summation.wrk_EventArraySize := 30;
END_DATA_BLOCK

DATA_BLOCK "Warning"   // DB31611
TITLE = CPG_Warning
{ S7_Optimized_Access := 'TRUE' }
AUTHOR : tech.team.motioncontrol@siemens.com
FAMILY : CPG
VERSION : 1.0
// Support: tech.team.motioncontrol@siemens.com
// Fax: +49 (0) 9131/98-1297
// stored: AutoNumber true, DBAccessibleFromOPCUA true, DBAccessibleFromWebserver true, IsOnlyStoredInLoadMemory false, IsRetainMemResEnabled false, IsWriteProtectedInAS false, MemoryReserve 0
   VAR
      Summation { ExternalWritable := 'False'; S7_SetPoint := 'True'} : "CPG_typeEventSummation";   // Unit Mode - Warning Summation
   END_VAR
BEGIN
   Summation.wrk_EventArraySize := 30;
END_DATA_BLOCK

DATA_BLOCK "UN"   // DB31629
TITLE = UN
{ S7_Optimized_Access := 'TRUE' }
AUTHOR : tech.team.motioncontrol@siemens.com
FAMILY : CPG
VERSION : 1.0
// Support: tech.team.motioncontrol@siemens.com
// Fax: +49 (0) 9131/98-1297
// stored: AutoNumber true, DBAccessibleFromOPCUA true, DBAccessibleFromWebserver true, IsOnlyStoredInLoadMemory false, IsRetainMemResEnabled false, IsWriteProtectedInAS false, MemoryReserve 100
   VAR
      PackML_Sts { ExternalWritable := 'False'; S7_SetPoint := 'True'} : "CPG_typePackML_ModuleSts";   // PackML Module Status - UN Status
      PackML_Sts_Alarm { ExternalWritable := 'False'; S7_SetPoint := 'True'} : "CPG_typePackML_ModuleSts";   // PackML Module Status - UN alarm status
      Alarm { ExternalAccessible := 'False'; ExternalVisible := 'False'; ExternalWritable := 'False'; S7_SetPoint := 'True'} : "CPG_typeEventStatus";   // Alarm Event Status - UN Status
      Warning { ExternalAccessible := 'False'; ExternalVisible := 'False'; ExternalWritable := 'False'; S7_SetPoint := 'True'} : "CPG_typeEventStatus";   // Warning Event Status - UN Status
      Status { ExternalAccessible := 'False'; ExternalVisible := 'False'; ExternalWritable := 'False'; S7_SetPoint := 'True'} : "CPG_typeEventStatus";   // Event Status - UN Status
   END_VAR
BEGIN
END_DATA_BLOCK

DATA_BLOCK "AlarmCfg"   // DB31600
TITLE = CPG_AlarmCfg
{ S7_Optimized_Access := 'TRUE' }
AUTHOR : tech.team.motioncontrol@siemens.com
FAMILY : CPG
VERSION : 1.0
// Support: tech.team.motioncontrol@siemens.com
// Fax: +49 (0) 9131/98-1297
// stored: AutoNumber true, DBAccessibleFromOPCUA true, DBAccessibleFromWebserver true, IsOnlyStoredInLoadMemory false, IsRetainMemResEnabled false, IsWriteProtectedInAS false, MemoryReserve 0
   VAR
      Event { ExternalAccessible := 'False'; ExternalVisible := 'False'; ExternalWritable := 'False'; S7_SetPoint := 'True'} : Array[0.."CPG_NO_OF_CFG_ALARMS_UPPER_LIM"] of "CPG_typeEventCfg";
   END_VAR
BEGIN
   // Event[0] : Alarm Test
   // Event[1] : Emergency Stop
   // Event[2] : Guard Door
   // Event[3] : Stop Command
   // Event[4] : Hold Command
   // Event[5] : Axis Error
   // Event[6] : Drive Fault
   // Event[7] : Machine Blocked
   // Event[8] : Machine Starved - No bottles
   // Event[9] : Machine Starved - No labels
   // Event[10] : Spare
   // Event[11] : Spare
   // Event[12] : Spare
   // Event[13] : Spare
   // Event[14] : Spare
   // Event[15] : Spare
   // Event[16] : Spare
   // Event[17] : Spare
   // Event[18] : Spare
   // Event[19] : Spare
   // Event[20] : Remote Stop Command
   // Event[21] : Remote Abort Command
   // Event[22] : Rmt Suspd Cmd - Blocked
   // Event[23] : Rmt Suspd Cmd - Starved
   // Event[24] : Remote Hold Cmd
   // Event[25] : Spare
   // Event[26] : Spare
   // Event[27] : Spare
   // Event[28] : Spare
   // Event[29] : Spare
   // Event[30] : Spare
   // Event[31] : Spare
   // Event[32] : Spare
   // Event[33] : Spare
   // Event[34] : Spare
   // Event[35] : Spare
   // Event[36] : Spare
   // Event[37] : Spare
   // Event[38] : Spare
   // Event[39] : Spare
   Event[0].ID := 0;
   Event[1].ID := 1;
   Event[2].ID := 4;
   Event[3].ID := 33;
   Event[4].ID := 40;
   Event[5].ID := 262;
   Event[6].ID := 261;
   Event[7].ID := 7;
   Event[8].ID := 8;
   Event[9].ID := 9;
   Event[20].ID := 41;
   Event[21].ID := 42;
   Event[22..23].ID := 43;
   Event[24].ID := 44;
   Event[1..2].value := 1;
   Event[3].value := 2;
   Event[4..5].value := 0;
   Event[6].value := 1;
   Event[7].value := 7;
   Event[8].value := 8;
   Event[9].value := 9;
   Event[20].value := 20;
   Event[21].value := 21;
   Event[22].value := 22;
   Event[23].value := 23;
   Event[24].value := 24;
   Event[38].value := 0;
   Event[0].message[0..2] := 'Alarm Test';
   Event[1].message[0] := 'E-Stop';
   Event[1].message[1] := 'Not-Halt';
   Event[1].message[2] := 'Los E-Stop';
   Event[2].message[0] := 'Guard Door';
   Event[2].message[1] := 'Schutzzaun';
   Event[2].message[2] := 'Las Guard Door';
   Event[3].message[0] := 'Stop PB';
   Event[3].message[1] := 'Stopp Taster';
   Event[3].message[2] := 'Las Stop PB';
   Event[4].message[0] := 'Hold PB';
   Event[4].message[1] := 'Hold Taster';
   Event[4].message[2] := 'Las Hold PB';
   Event[5].message[0] := 'Axis Error';
   Event[5].message[1] := 'Achsfehler';
   Event[5].message[2] := 'Las Axis Error';
   Event[6].message[0] := 'Drive Faulted';
   Event[6].message[1] := 'Antriebsfehler';
   Event[6].message[2] := 'Los Drive Faulted';
   Event[7].message[0] := 'Machine Blocked';
   Event[7].message[1] := 'Maschine blockiert';
   Event[7].message[2] := 'Los Machine Blocked';
   Event[8].message[0] := 'Starved - No botttles';
   Event[8].message[1] := 'Flaschenzufuhr leer';
   Event[8].message[2] := 'Las Starved - No botttles';
   Event[9].message[0] := 'Starved - No labels';
   Event[9].message[1] := 'Etikettenzufuhr leer';
   Event[9].message[2] := 'Las Starved - No labels';
   Event[10].message[0] := 'Spare';
   Event[10].message[1] := 'Reserve';
   Event[10].message[2] := 'Spare';
   Event[11].message[0] := 'Spare';
   Event[11].message[1] := 'Reserve';
   Event[11].message[2] := 'Spare';
   Event[12].message[0] := 'Spare';
   Event[12].message[1] := 'Reserve';
   Event[12].message[2] := 'Spare';
   Event[13].message[0] := 'Spare';
   Event[13].message[1] := 'Reserve';
   Event[13].message[2] := 'Spare';
   Event[14].message[0] := 'Spare';
   Event[14].message[1] := 'Reserve';
   Event[14].message[2] := 'Spare';
   Event[15].message[0] := 'Spare';
   Event[15].message[1] := 'Reserve';
   Event[15].message[2] := 'Spare';
   Event[16].message[0] := 'Spare';
   Event[16].message[1] := 'Reserve';
   Event[16].message[2] := 'Spare';
   Event[17].message[0] := 'Spare';
   Event[17].message[1] := 'Reserve';
   Event[17].message[2] := 'Spare';
   Event[18].message[0] := 'Spare';
   Event[18].message[1] := 'Reserve';
   Event[18].message[2] := 'Spare';
   Event[19].message[0] := 'Spare';
   Event[19].message[1] := 'Reserve';
   Event[19].message[2] := 'Spare';
   Event[20].message[0..1] := 'Remote Stop Cmd';
   Event[20].message[2] := 'Las Remote Stop Cmd';
   Event[21].message[0..1] := 'Remote Abort Cmd';
   Event[21].message[2] := 'Las Remote Abort Cmd';
   Event[22].message[0] := 'Rmt Suspd Cmd - Blocked';
   Event[22].message[1] := 'Remote Suspend Cmd - Blocked';
   Event[22].message[2] := 'Las Remote Suspd Cmd - Blocked';
   Event[23].message[0] := 'Rmt Suspd Cmd - Starved';
   Event[23].message[1] := 'Remote Suspend Cmd - Starved';
   Event[23].message[2] := 'Las Rmt Suspd Cmd - Starved';
   Event[24].message[0..1] := 'Remote Hold Cmd';
   Event[24].message[2] := 'Las Remote Hold Cmd';
   Event[25].message[0] := 'Spare';
   Event[25].message[1] := 'Reserve';
   Event[25].message[2] := 'Spare';
   Event[26].message[0] := 'Spare';
   Event[26].message[1] := 'Reserve';
   Event[26].message[2] := 'Spare';
   Event[27].message[0] := 'Spare';
   Event[27].message[1] := 'Reserve';
   Event[27].message[2] := 'Spare';
   Event[28].message[0] := 'Spare';
   Event[28].message[1] := 'Reserve';
   Event[28].message[2] := 'Spare';
   Event[29].message[0] := 'Spare';
   Event[29].message[1] := 'Reserve';
   Event[29].message[2] := 'Spare';
   Event[30].message[0] := 'Spare';
   Event[30].message[1] := 'Reserve';
   Event[30].message[2] := 'Spare';
   Event[31].message[0] := 'Spare';
   Event[31].message[1] := 'Reserve';
   Event[31].message[2] := 'Spare';
   Event[32].message[0] := 'Spare';
   Event[32].message[1] := 'Reserve';
   Event[32].message[2] := 'Spare';
   Event[33].message[0] := 'Spare';
   Event[33].message[1] := 'Reserve';
   Event[33].message[2] := 'Spare';
   Event[34].message[0] := 'Spare';
   Event[34].message[1] := 'Reserve';
   Event[34].message[2] := 'Spare';
   Event[35].message[0] := 'Spare';
   Event[35].message[1] := 'Reserve';
   Event[35].message[2] := 'Spare';
   Event[36].message[0] := 'Spare';
   Event[36].message[1] := 'Reserve';
   Event[36].message[2] := 'Spare';
   Event[37].message[0] := 'Spare';
   Event[37].message[1] := 'Reserve';
   Event[37].message[2] := 'Spare';
   Event[38].message[0] := 'Spare';
   Event[38].message[1] := 'Reserve';
   Event[38].message[2] := 'Spare';
   Event[39].message[0] := 'Spare';
   Event[39].message[1] := 'Reserve';
   Event[39].message[2] := 'Spare';
   Event[0].category := 6;
   Event[1].category := 0;   // 0 = Safety related, Coordinated fast stop
   // Event[2].category : 0 = Safety related, Coordinated fast stop
   Event[3].category := 2;   // 2 = Coordinated normal stop
   Event[4].category := 7;   // 7 = Held command
   Event[5].category := 1;   // 1 = Coordinated fast stop
   Event[6].category := 1;   // 1 = Coordinated fast stop
   Event[7].category := 8;   // 8 =Blocked, Coordinated slow stop
   Event[8].category := 9;   // 9 = Starved, Coordinated slow stop
   Event[9].category := 9;   // 9 = Starved, Coordinated slow stop
   Event[10].category := 0;   // 9 = Starved, Coordinated slow stop
   Event[11..13].category := 0;
   Event[20].category := 2;   // 2 = Coordinated normal stop
   Event[21].category := 1;   // 0 = Safety related, Coordinated fast stop
   Event[22].category := 8;   // 9 = Starved, Coordinated slow stop
   Event[23].category := 9;   // 7 = Hold, Coordinated slow stop
   Event[24].category := 7;   // 7 = Coordinated slow stop
END_DATA_BLOCK

DATA_BLOCK "MessagePrefix"   // DB31604
TITLE = CPG_MessagePrefix
{ S7_Optimized_Access := 'TRUE' }
AUTHOR : tech.team.motioncontrol@siemens.com
FAMILY : CPG
VERSION : 1.0
// Support: tech.team.motioncontrol@siemens.com
// Fax: +49 (0) 9131/98-1297
// stored: AutoNumber true, DBAccessibleFromOPCUA true, DBAccessibleFromWebserver true, IsOnlyStoredInLoadMemory false, IsRetainMemResEnabled false, IsWriteProtectedInAS false, MemoryReserve 0
   VAR
      UN { ExternalAccessible := 'False'; ExternalVisible := 'False'; ExternalWritable := 'False'} : Struct   // MessagePrefix for Unit
         Alarm { ExternalAccessible := 'False'; ExternalVisible := 'False'; ExternalWritable := 'False'; S7_SetPoint := 'True'} : "CPG_typeMessagePrefix";   // MessagePrefix for Unit Alarms
      END_STRUCT;
      EM00 { ExternalAccessible := 'False'; ExternalVisible := 'False'; ExternalWritable := 'False'} : Struct   // MessagePrefix for EquipmentModuleEM00
         EventControl { ExternalAccessible := 'False'; ExternalVisible := 'False'; ExternalWritable := 'False'; S7_SetPoint := 'True'} : "CPG_typeMessagePrefix";   // MessagePrefixforEventControl
         CM01 { ExternalAccessible := 'False'; ExternalVisible := 'False'; ExternalWritable := 'False'; S7_SetPoint := 'True'} : "CPG_typeMessagePrefix";   // MessagePrefixforControlModule#01
         CM02 { ExternalAccessible := 'False'; ExternalVisible := 'False'; ExternalWritable := 'False'; S7_SetPoint := 'True'} : "CPG_typeMessagePrefix";   // MessagePrefixforControlModule#02
         CM03 { ExternalAccessible := 'False'; ExternalVisible := 'False'; ExternalWritable := 'False'; S7_SetPoint := 'True'} : "CPG_typeMessagePrefix";   // MessagePrefixforControlModule#03
         CM04 { ExternalAccessible := 'False'; ExternalVisible := 'False'; ExternalWritable := 'False'; S7_SetPoint := 'True'} : "CPG_typeMessagePrefix";   // MessagePrefixforControlModule#04
         CM05 { ExternalAccessible := 'False'; ExternalVisible := 'False'; ExternalWritable := 'False'; S7_SetPoint := 'True'} : "CPG_typeMessagePrefix";   // MessagePrefixforControlModule#05
         CM06 { ExternalAccessible := 'False'; ExternalVisible := 'False'; ExternalWritable := 'False'; S7_SetPoint := 'True'} : "CPG_typeMessagePrefix";   // MessagePrefixforControlModule#06
         CM07 { ExternalAccessible := 'False'; ExternalVisible := 'False'; ExternalWritable := 'False'; S7_SetPoint := 'True'} : "CPG_typeMessagePrefix";   // MessagePrefixforControlModule#07
         CM08 { ExternalAccessible := 'False'; ExternalVisible := 'False'; ExternalWritable := 'False'; S7_SetPoint := 'True'} : "CPG_typeMessagePrefix";   // MessagePrefixforControlModule#08
         CM09 { ExternalAccessible := 'False'; ExternalVisible := 'False'; ExternalWritable := 'False'; S7_SetPoint := 'True'} : "CPG_typeMessagePrefix";   // MessagePrefixforControlModule#09
         CM10 { ExternalAccessible := 'False'; ExternalVisible := 'False'; ExternalWritable := 'False'; S7_SetPoint := 'True'} : "CPG_typeMessagePrefix";   // MessagePrefixforControlModule#10
      END_STRUCT;
      EM01 { ExternalAccessible := 'False'; ExternalVisible := 'False'; ExternalWritable := 'False'} : Struct   // MessagePrefix for EquipmentModuleEM01
         EventControl { ExternalAccessible := 'False'; ExternalVisible := 'False'; ExternalWritable := 'False'; S7_SetPoint := 'True'} : "CPG_typeMessagePrefix";   // MessagePrefixforEventControl
         CM01 { ExternalAccessible := 'False'; ExternalVisible := 'False'; ExternalWritable := 'False'; S7_SetPoint := 'True'} : "CPG_typeMessagePrefix";   // MessagePrefixforControlModule#01
         CM02 { ExternalAccessible := 'False'; ExternalVisible := 'False'; ExternalWritable := 'False'; S7_SetPoint := 'True'} : "CPG_typeMessagePrefix";   // MessagePrefixforControlModule#02
         CM03 { ExternalAccessible := 'False'; ExternalVisible := 'False'; ExternalWritable := 'False'; S7_SetPoint := 'True'} : "CPG_typeMessagePrefix";   // MessagePrefixforControlModule#03
         CM04 { ExternalAccessible := 'False'; ExternalVisible := 'False'; ExternalWritable := 'False'; S7_SetPoint := 'True'} : "CPG_typeMessagePrefix";   // MessagePrefixforControlModule#04
         CM05 { ExternalAccessible := 'False'; ExternalVisible := 'False'; ExternalWritable := 'False'; S7_SetPoint := 'True'} : "CPG_typeMessagePrefix";   // MessagePrefixforControlModule#05
         CM06 { ExternalAccessible := 'False'; ExternalVisible := 'False'; ExternalWritable := 'False'; S7_SetPoint := 'True'} : "CPG_typeMessagePrefix";   // MessagePrefixforControlModule#06
         CM07 { ExternalAccessible := 'False'; ExternalVisible := 'False'; ExternalWritable := 'False'; S7_SetPoint := 'True'} : "CPG_typeMessagePrefix";   // MessagePrefixforControlModule#07
         CM08 { ExternalAccessible := 'False'; ExternalVisible := 'False'; ExternalWritable := 'False'; S7_SetPoint := 'True'} : "CPG_typeMessagePrefix";   // MessagePrefixforControlModule#08
         CM09 { ExternalAccessible := 'False'; ExternalVisible := 'False'; ExternalWritable := 'False'; S7_SetPoint := 'True'} : "CPG_typeMessagePrefix";   // MessagePrefixforControlModule#09
         CM10 { ExternalAccessible := 'False'; ExternalVisible := 'False'; ExternalWritable := 'False'; S7_SetPoint := 'True'} : "CPG_typeMessagePrefix";   // MessagePrefixforControlModule#10
      END_STRUCT;
      EM02 { ExternalAccessible := 'False'; ExternalVisible := 'False'; ExternalWritable := 'False'} : Struct   // MessagePrefix for EquipmentModuleEM02
         EventControl { ExternalAccessible := 'False'; ExternalVisible := 'False'; ExternalWritable := 'False'; S7_SetPoint := 'True'} : "CPG_typeMessagePrefix";   // MessagePrefixforEventControl
         CM01 { ExternalAccessible := 'False'; ExternalVisible := 'False'; ExternalWritable := 'False'; S7_SetPoint := 'True'} : "CPG_typeMessagePrefix";   // MessagePrefixforControlModule#01
         CM02 { ExternalAccessible := 'False'; ExternalVisible := 'False'; ExternalWritable := 'False'; S7_SetPoint := 'True'} : "CPG_typeMessagePrefix";   // MessagePrefixforControlModule#02
         CM03 { ExternalAccessible := 'False'; ExternalVisible := 'False'; ExternalWritable := 'False'; S7_SetPoint := 'True'} : "CPG_typeMessagePrefix";   // MessagePrefixforControlModule#03
         CM04 { ExternalAccessible := 'False'; ExternalVisible := 'False'; ExternalWritable := 'False'; S7_SetPoint := 'True'} : "CPG_typeMessagePrefix";   // MessagePrefixforControlModule#04
         CM05 { ExternalAccessible := 'False'; ExternalVisible := 'False'; ExternalWritable := 'False'; S7_SetPoint := 'True'} : "CPG_typeMessagePrefix";   // MessagePrefixforControlModule#05
         CM06 { ExternalAccessible := 'False'; ExternalVisible := 'False'; ExternalWritable := 'False'; S7_SetPoint := 'True'} : "CPG_typeMessagePrefix";   // MessagePrefixforControlModule#06
         CM07 { ExternalAccessible := 'False'; ExternalVisible := 'False'; ExternalWritable := 'False'; S7_SetPoint := 'True'} : "CPG_typeMessagePrefix";   // MessagePrefixforControlModule#07
         CM08 { ExternalAccessible := 'False'; ExternalVisible := 'False'; ExternalWritable := 'False'; S7_SetPoint := 'True'} : "CPG_typeMessagePrefix";   // MessagePrefixforControlModule#08
         CM09 { ExternalAccessible := 'False'; ExternalVisible := 'False'; ExternalWritable := 'False'; S7_SetPoint := 'True'} : "CPG_typeMessagePrefix";   // MessagePrefixforControlModule#09
         CM10 { ExternalAccessible := 'False'; ExternalVisible := 'False'; ExternalWritable := 'False'; S7_SetPoint := 'True'} : "CPG_typeMessagePrefix";   // MessagePrefixforControlModule#10
      END_STRUCT;
      EM03 { ExternalAccessible := 'False'; ExternalVisible := 'False'; ExternalWritable := 'False'} : Struct   // MessagePrefix for EquipmentModuleEM03
         EventControl { ExternalAccessible := 'False'; ExternalVisible := 'False'; ExternalWritable := 'False'; S7_SetPoint := 'True'} : "CPG_typeMessagePrefix";   // MessagePrefixforEventControl
         CM01 { ExternalAccessible := 'False'; ExternalVisible := 'False'; ExternalWritable := 'False'; S7_SetPoint := 'True'} : "CPG_typeMessagePrefix";   // MessagePrefixforControlModule#01
         CM02 { ExternalAccessible := 'False'; ExternalVisible := 'False'; ExternalWritable := 'False'; S7_SetPoint := 'True'} : "CPG_typeMessagePrefix";   // MessagePrefixforControlModule#02
         CM03 { ExternalAccessible := 'False'; ExternalVisible := 'False'; ExternalWritable := 'False'; S7_SetPoint := 'True'} : "CPG_typeMessagePrefix";   // MessagePrefixforControlModule#03
         CM04 { ExternalAccessible := 'False'; ExternalVisible := 'False'; ExternalWritable := 'False'; S7_SetPoint := 'True'} : "CPG_typeMessagePrefix";   // MessagePrefixforControlModule#04
         CM05 { ExternalAccessible := 'False'; ExternalVisible := 'False'; ExternalWritable := 'False'; S7_SetPoint := 'True'} : "CPG_typeMessagePrefix";   // MessagePrefixforControlModule#05
         CM06 { ExternalAccessible := 'False'; ExternalVisible := 'False'; ExternalWritable := 'False'; S7_SetPoint := 'True'} : "CPG_typeMessagePrefix";   // MessagePrefixforControlModule#06
         CM07 { ExternalAccessible := 'False'; ExternalVisible := 'False'; ExternalWritable := 'False'; S7_SetPoint := 'True'} : "CPG_typeMessagePrefix";   // MessagePrefixforControlModule#07
         CM08 { ExternalAccessible := 'False'; ExternalVisible := 'False'; ExternalWritable := 'False'; S7_SetPoint := 'True'} : "CPG_typeMessagePrefix";   // MessagePrefixforControlModule#08
         CM09 { ExternalAccessible := 'False'; ExternalVisible := 'False'; ExternalWritable := 'False'; S7_SetPoint := 'True'} : "CPG_typeMessagePrefix";   // MessagePrefixforControlModule#09
         CM10 { ExternalAccessible := 'False'; ExternalVisible := 'False'; ExternalWritable := 'False'; S7_SetPoint := 'True'} : "CPG_typeMessagePrefix";   // MessagePrefixforControlModule#10
      END_STRUCT;
      EM04 { ExternalAccessible := 'False'; ExternalVisible := 'False'; ExternalWritable := 'False'} : Struct   // MessagePrefix for EquipmentModuleEM04
         EventControl { ExternalAccessible := 'False'; ExternalVisible := 'False'; ExternalWritable := 'False'; S7_SetPoint := 'True'} : "CPG_typeMessagePrefix";   // MessagePrefixforEventControl
         CM01 { ExternalAccessible := 'False'; ExternalVisible := 'False'; ExternalWritable := 'False'; S7_SetPoint := 'True'} : "CPG_typeMessagePrefix";   // MessagePrefixforControlModule#01
         CM02 { ExternalAccessible := 'False'; ExternalVisible := 'False'; ExternalWritable := 'False'; S7_SetPoint := 'True'} : "CPG_typeMessagePrefix";   // MessagePrefixforControlModule#02
         CM03 { ExternalAccessible := 'False'; ExternalVisible := 'False'; ExternalWritable := 'False'; S7_SetPoint := 'True'} : "CPG_typeMessagePrefix";   // MessagePrefixforControlModule#03
         CM04 { ExternalAccessible := 'False'; ExternalVisible := 'False'; ExternalWritable := 'False'; S7_SetPoint := 'True'} : "CPG_typeMessagePrefix";   // MessagePrefixforControlModule#04
         CM05 { ExternalAccessible := 'False'; ExternalVisible := 'False'; ExternalWritable := 'False'; S7_SetPoint := 'True'} : "CPG_typeMessagePrefix";   // MessagePrefixforControlModule#05
         CM06 { ExternalAccessible := 'False'; ExternalVisible := 'False'; ExternalWritable := 'False'; S7_SetPoint := 'True'} : "CPG_typeMessagePrefix";   // MessagePrefixforControlModule#06
         CM07 { ExternalAccessible := 'False'; ExternalVisible := 'False'; ExternalWritable := 'False'; S7_SetPoint := 'True'} : "CPG_typeMessagePrefix";   // MessagePrefixforControlModule#07
         CM08 { ExternalAccessible := 'False'; ExternalVisible := 'False'; ExternalWritable := 'False'; S7_SetPoint := 'True'} : "CPG_typeMessagePrefix";   // MessagePrefixforControlModule#08
         CM09 { ExternalAccessible := 'False'; ExternalVisible := 'False'; ExternalWritable := 'False'; S7_SetPoint := 'True'} : "CPG_typeMessagePrefix";   // MessagePrefixforControlModule#09
         CM10 { ExternalAccessible := 'False'; ExternalVisible := 'False'; ExternalWritable := 'False'; S7_SetPoint := 'True'} : "CPG_typeMessagePrefix";   // MessagePrefixforControlModule#10
      END_STRUCT;
      EM05 { ExternalAccessible := 'False'; ExternalVisible := 'False'; ExternalWritable := 'False'} : Struct   // MessagePrefix for EquipmentModuleEM05
         EventControl { ExternalAccessible := 'False'; ExternalVisible := 'False'; ExternalWritable := 'False'; S7_SetPoint := 'True'} : "CPG_typeMessagePrefix";   // MessagePrefixforEventControl
         CM01 { ExternalAccessible := 'False'; ExternalVisible := 'False'; ExternalWritable := 'False'; S7_SetPoint := 'True'} : "CPG_typeMessagePrefix";   // MessagePrefixforControlModule#01
         CM02 { ExternalAccessible := 'False'; ExternalVisible := 'False'; ExternalWritable := 'False'; S7_SetPoint := 'True'} : "CPG_typeMessagePrefix";   // MessagePrefixforControlModule#02
         CM03 { ExternalAccessible := 'False'; ExternalVisible := 'False'; ExternalWritable := 'False'; S7_SetPoint := 'True'} : "CPG_typeMessagePrefix";   // MessagePrefixforControlModule#03
         CM04 { ExternalAccessible := 'False'; ExternalVisible := 'False'; ExternalWritable := 'False'; S7_SetPoint := 'True'} : "CPG_typeMessagePrefix";   // MessagePrefixforControlModule#04
         CM05 { ExternalAccessible := 'False'; ExternalVisible := 'False'; ExternalWritable := 'False'; S7_SetPoint := 'True'} : "CPG_typeMessagePrefix";   // MessagePrefixforControlModule#05
         CM06 { ExternalAccessible := 'False'; ExternalVisible := 'False'; ExternalWritable := 'False'; S7_SetPoint := 'True'} : "CPG_typeMessagePrefix";   // MessagePrefixforControlModule#06
         CM07 { ExternalAccessible := 'False'; ExternalVisible := 'False'; ExternalWritable := 'False'; S7_SetPoint := 'True'} : "CPG_typeMessagePrefix";   // MessagePrefixforControlModule#07
         CM08 { ExternalAccessible := 'False'; ExternalVisible := 'False'; ExternalWritable := 'False'; S7_SetPoint := 'True'} : "CPG_typeMessagePrefix";   // MessagePrefixforControlModule#08
         CM09 { ExternalAccessible := 'False'; ExternalVisible := 'False'; ExternalWritable := 'False'; S7_SetPoint := 'True'} : "CPG_typeMessagePrefix";   // MessagePrefixforControlModule#09
         CM10 { ExternalAccessible := 'False'; ExternalVisible := 'False'; ExternalWritable := 'False'; S7_SetPoint := 'True'} : "CPG_typeMessagePrefix";   // MessagePrefixforControlModule#10
      END_STRUCT;
      EM06 { ExternalAccessible := 'False'; ExternalVisible := 'False'; ExternalWritable := 'False'} : Struct   // MessagePrefix for EquipmentModuleEM06
         EventControl { ExternalAccessible := 'False'; ExternalVisible := 'False'; ExternalWritable := 'False'; S7_SetPoint := 'True'} : "CPG_typeMessagePrefix";   // MessagePrefixforEventControl
         CM01 { ExternalAccessible := 'False'; ExternalVisible := 'False'; ExternalWritable := 'False'; S7_SetPoint := 'True'} : "CPG_typeMessagePrefix";   // MessagePrefixforControlModule#01
         CM02 { ExternalAccessible := 'False'; ExternalVisible := 'False'; ExternalWritable := 'False'; S7_SetPoint := 'True'} : "CPG_typeMessagePrefix";   // MessagePrefixforControlModule#02
         CM03 { ExternalAccessible := 'False'; ExternalVisible := 'False'; ExternalWritable := 'False'; S7_SetPoint := 'True'} : "CPG_typeMessagePrefix";   // MessagePrefixforControlModule#03
         CM04 { ExternalAccessible := 'False'; ExternalVisible := 'False'; ExternalWritable := 'False'; S7_SetPoint := 'True'} : "CPG_typeMessagePrefix";   // MessagePrefixforControlModule#04
         CM05 { ExternalAccessible := 'False'; ExternalVisible := 'False'; ExternalWritable := 'False'; S7_SetPoint := 'True'} : "CPG_typeMessagePrefix";   // MessagePrefixforControlModule#05
         CM06 { ExternalAccessible := 'False'; ExternalVisible := 'False'; ExternalWritable := 'False'; S7_SetPoint := 'True'} : "CPG_typeMessagePrefix";   // MessagePrefixforControlModule#06
         CM07 { ExternalAccessible := 'False'; ExternalVisible := 'False'; ExternalWritable := 'False'; S7_SetPoint := 'True'} : "CPG_typeMessagePrefix";   // MessagePrefixforControlModule#07
         CM08 { ExternalAccessible := 'False'; ExternalVisible := 'False'; ExternalWritable := 'False'; S7_SetPoint := 'True'} : "CPG_typeMessagePrefix";   // MessagePrefixforControlModule#08
         CM09 { ExternalAccessible := 'False'; ExternalVisible := 'False'; ExternalWritable := 'False'; S7_SetPoint := 'True'} : "CPG_typeMessagePrefix";   // MessagePrefixforControlModule#09
         CM10 { ExternalAccessible := 'False'; ExternalVisible := 'False'; ExternalWritable := 'False'; S7_SetPoint := 'True'} : "CPG_typeMessagePrefix";   // MessagePrefixforControlModule#10
      END_STRUCT;
      EM07 { ExternalAccessible := 'False'; ExternalVisible := 'False'; ExternalWritable := 'False'} : Struct   // MessagePrefix for EquipmentModuleEM07
         EventControl { ExternalAccessible := 'False'; ExternalVisible := 'False'; ExternalWritable := 'False'; S7_SetPoint := 'True'} : "CPG_typeMessagePrefix";   // MessagePrefixforEventControl
         CM01 { ExternalAccessible := 'False'; ExternalVisible := 'False'; ExternalWritable := 'False'; S7_SetPoint := 'True'} : "CPG_typeMessagePrefix";   // MessagePrefixforControlModule#01
         CM02 { ExternalAccessible := 'False'; ExternalVisible := 'False'; ExternalWritable := 'False'; S7_SetPoint := 'True'} : "CPG_typeMessagePrefix";   // MessagePrefixforControlModule#02
         CM03 { ExternalAccessible := 'False'; ExternalVisible := 'False'; ExternalWritable := 'False'; S7_SetPoint := 'True'} : "CPG_typeMessagePrefix";   // MessagePrefixforControlModule#03
         CM04 { ExternalAccessible := 'False'; ExternalVisible := 'False'; ExternalWritable := 'False'; S7_SetPoint := 'True'} : "CPG_typeMessagePrefix";   // MessagePrefixforControlModule#04
         CM05 { ExternalAccessible := 'False'; ExternalVisible := 'False'; ExternalWritable := 'False'; S7_SetPoint := 'True'} : "CPG_typeMessagePrefix";   // MessagePrefixforControlModule#05
         CM06 { ExternalAccessible := 'False'; ExternalVisible := 'False'; ExternalWritable := 'False'; S7_SetPoint := 'True'} : "CPG_typeMessagePrefix";   // MessagePrefixforControlModule#06
         CM07 { ExternalAccessible := 'False'; ExternalVisible := 'False'; ExternalWritable := 'False'; S7_SetPoint := 'True'} : "CPG_typeMessagePrefix";   // MessagePrefixforControlModule#07
         CM08 { ExternalAccessible := 'False'; ExternalVisible := 'False'; ExternalWritable := 'False'; S7_SetPoint := 'True'} : "CPG_typeMessagePrefix";   // MessagePrefixforControlModule#08
         CM09 { ExternalAccessible := 'False'; ExternalVisible := 'False'; ExternalWritable := 'False'; S7_SetPoint := 'True'} : "CPG_typeMessagePrefix";   // MessagePrefixforControlModule#09
         CM10 { ExternalAccessible := 'False'; ExternalVisible := 'False'; ExternalWritable := 'False'; S7_SetPoint := 'True'} : "CPG_typeMessagePrefix";   // MessagePrefixforControlModule#10
      END_STRUCT;
      EM08 { ExternalAccessible := 'False'; ExternalVisible := 'False'; ExternalWritable := 'False'} : Struct   // MessagePrefix for EquipmentModuleEM08
         EventControl { ExternalAccessible := 'False'; ExternalVisible := 'False'; ExternalWritable := 'False'; S7_SetPoint := 'True'} : "CPG_typeMessagePrefix";   // MessagePrefixforEventControl
         CM01 { ExternalAccessible := 'False'; ExternalVisible := 'False'; ExternalWritable := 'False'; S7_SetPoint := 'True'} : "CPG_typeMessagePrefix";   // MessagePrefixforControlModule#01
         CM02 { ExternalAccessible := 'False'; ExternalVisible := 'False'; ExternalWritable := 'False'; S7_SetPoint := 'True'} : "CPG_typeMessagePrefix";   // MessagePrefixforControlModule#02
         CM03 { ExternalAccessible := 'False'; ExternalVisible := 'False'; ExternalWritable := 'False'; S7_SetPoint := 'True'} : "CPG_typeMessagePrefix";   // MessagePrefixforControlModule#03
         CM04 { ExternalAccessible := 'False'; ExternalVisible := 'False'; ExternalWritable := 'False'; S7_SetPoint := 'True'} : "CPG_typeMessagePrefix";   // MessagePrefixforControlModule#04
         CM05 { ExternalAccessible := 'False'; ExternalVisible := 'False'; ExternalWritable := 'False'; S7_SetPoint := 'True'} : "CPG_typeMessagePrefix";   // MessagePrefixforControlModule#05
         CM06 { ExternalAccessible := 'False'; ExternalVisible := 'False'; ExternalWritable := 'False'; S7_SetPoint := 'True'} : "CPG_typeMessagePrefix";   // MessagePrefixforControlModule#06
         CM07 { ExternalAccessible := 'False'; ExternalVisible := 'False'; ExternalWritable := 'False'; S7_SetPoint := 'True'} : "CPG_typeMessagePrefix";   // MessagePrefixforControlModule#07
         CM08 { ExternalAccessible := 'False'; ExternalVisible := 'False'; ExternalWritable := 'False'; S7_SetPoint := 'True'} : "CPG_typeMessagePrefix";   // MessagePrefixforControlModule#08
         CM09 { ExternalAccessible := 'False'; ExternalVisible := 'False'; ExternalWritable := 'False'; S7_SetPoint := 'True'} : "CPG_typeMessagePrefix";   // MessagePrefixforControlModule#09
         CM10 { ExternalAccessible := 'False'; ExternalVisible := 'False'; ExternalWritable := 'False'; S7_SetPoint := 'True'} : "CPG_typeMessagePrefix";   // MessagePrefixforControlModule#10
      END_STRUCT;
      EM09 { ExternalAccessible := 'False'; ExternalVisible := 'False'; ExternalWritable := 'False'} : Struct   // MessagePrefix for EquipmentModuleEM09
         EventControl { ExternalAccessible := 'False'; ExternalVisible := 'False'; ExternalWritable := 'False'; S7_SetPoint := 'True'} : "CPG_typeMessagePrefix";   // MessagePrefixforEventControl
         CM01 { ExternalAccessible := 'False'; ExternalVisible := 'False'; ExternalWritable := 'False'; S7_SetPoint := 'True'} : "CPG_typeMessagePrefix";   // MessagePrefixforControlModule#01
         CM02 { ExternalAccessible := 'False'; ExternalVisible := 'False'; ExternalWritable := 'False'; S7_SetPoint := 'True'} : "CPG_typeMessagePrefix";   // MessagePrefixforControlModule#02
         CM03 { ExternalAccessible := 'False'; ExternalVisible := 'False'; ExternalWritable := 'False'; S7_SetPoint := 'True'} : "CPG_typeMessagePrefix";   // MessagePrefixforControlModule#03
         CM04 { ExternalAccessible := 'False'; ExternalVisible := 'False'; ExternalWritable := 'False'; S7_SetPoint := 'True'} : "CPG_typeMessagePrefix";   // MessagePrefixforControlModule#04
         CM05 { ExternalAccessible := 'False'; ExternalVisible := 'False'; ExternalWritable := 'False'; S7_SetPoint := 'True'} : "CPG_typeMessagePrefix";   // MessagePrefixforControlModule#05
         CM06 { ExternalAccessible := 'False'; ExternalVisible := 'False'; ExternalWritable := 'False'; S7_SetPoint := 'True'} : "CPG_typeMessagePrefix";   // MessagePrefixforControlModule#06
         CM07 { ExternalAccessible := 'False'; ExternalVisible := 'False'; ExternalWritable := 'False'; S7_SetPoint := 'True'} : "CPG_typeMessagePrefix";   // MessagePrefixforControlModule#07
         CM08 { ExternalAccessible := 'False'; ExternalVisible := 'False'; ExternalWritable := 'False'; S7_SetPoint := 'True'} : "CPG_typeMessagePrefix";   // MessagePrefixforControlModule#08
         CM09 { ExternalAccessible := 'False'; ExternalVisible := 'False'; ExternalWritable := 'False'; S7_SetPoint := 'True'} : "CPG_typeMessagePrefix";   // MessagePrefixforControlModule#09
         CM10 { ExternalAccessible := 'False'; ExternalVisible := 'False'; ExternalWritable := 'False'; S7_SetPoint := 'True'} : "CPG_typeMessagePrefix";   // MessagePrefixforControlModule#10
      END_STRUCT;
   END_VAR
BEGIN
   UN.Alarm.messagePrefix[0..2] := 'Unit ';
   EM00.EventControl.messagePrefix[0..2] := 'EM00 ';
   EM00.CM01.messagePrefix[0..2] := 'CM01 ';
   EM00.CM02.messagePrefix[0..2] := 'CM02 ';
   EM00.CM03.messagePrefix[0..2] := 'CM03 ';
   EM00.CM04.messagePrefix[0..2] := 'CM04 ';
   EM00.CM05.messagePrefix[0..2] := 'CM05 ';
   EM00.CM06.messagePrefix[0..2] := 'CM06 ';
   EM00.CM07.messagePrefix[0..2] := 'CM07 ';
   EM00.CM08.messagePrefix[0..2] := 'CM08 ';
   EM00.CM09.messagePrefix[0..2] := 'CM09 ';
   EM00.CM10.messagePrefix[0..2] := 'CM10 ';
   EM01.EventControl.messagePrefix[0..2] := 'EM01 ';
   EM01.CM01.messagePrefix[0..2] := 'CM01 ';
   EM01.CM02.messagePrefix[0..2] := 'CM02 ';
   EM01.CM03.messagePrefix[0..2] := 'CM03 ';
   EM01.CM04.messagePrefix[0..2] := 'CM04 ';
   EM01.CM05.messagePrefix[0..2] := 'CM05 ';
   EM01.CM06.messagePrefix[0..2] := 'CM06 ';
   EM01.CM07.messagePrefix[0..2] := 'CM07 ';
   EM01.CM08.messagePrefix[0..2] := 'CM08 ';
   EM01.CM09.messagePrefix[0..2] := 'CM09 ';
   EM01.CM10.messagePrefix[0..2] := 'CM10 ';
   EM02.EventControl.messagePrefix[0..2] := 'EM01 ';
   EM02.CM01.messagePrefix[0..2] := 'CM01 ';
   EM02.CM02.messagePrefix[0..2] := 'CM02 ';
   EM02.CM03.messagePrefix[0..2] := 'CM03 ';
   EM02.CM04.messagePrefix[0..2] := 'CM04 ';
   EM02.CM05.messagePrefix[0..2] := 'CM05 ';
   EM02.CM06.messagePrefix[0..2] := 'CM06 ';
   EM02.CM07.messagePrefix[0..2] := 'CM07 ';
   EM02.CM08.messagePrefix[0..2] := 'CM08 ';
   EM02.CM09.messagePrefix[0..2] := 'CM09 ';
   EM02.CM10.messagePrefix[0..2] := 'CM10 ';
   EM03.EventControl.messagePrefix[0..2] := 'EM03 ';
   EM03.CM01.messagePrefix[0..2] := 'CM01 ';
   EM03.CM02.messagePrefix[0..2] := 'CM02 ';
   EM03.CM03.messagePrefix[0..2] := 'CM03 ';
   EM03.CM04.messagePrefix[0..2] := 'CM04 ';
   EM03.CM05.messagePrefix[0..2] := 'CM05 ';
   EM03.CM06.messagePrefix[0..2] := 'CM06 ';
   EM03.CM07.messagePrefix[0..2] := 'CM07 ';
   EM03.CM08.messagePrefix[0..2] := 'CM08 ';
   EM03.CM09.messagePrefix[0..2] := 'CM09 ';
   EM03.CM10.messagePrefix[0..2] := 'CM10 ';
   EM04.EventControl.messagePrefix[0..2] := 'EM04 ';
   EM04.CM01.messagePrefix[0..2] := 'CM01 ';
   EM04.CM02.messagePrefix[0..2] := 'CM02 ';
   EM04.CM03.messagePrefix[0..2] := 'CM03 ';
   EM04.CM04.messagePrefix[0..2] := 'CM04 ';
   EM04.CM05.messagePrefix[0..2] := 'CM05 ';
   EM04.CM06.messagePrefix[0..2] := 'CM06 ';
   EM04.CM07.messagePrefix[0..2] := 'CM07 ';
   EM04.CM08.messagePrefix[0..2] := 'CM08 ';
   EM04.CM09.messagePrefix[0..2] := 'CM09 ';
   EM04.CM10.messagePrefix[0..2] := 'CM10 ';
   EM05.EventControl.messagePrefix[0..2] := 'EM05 ';
   EM05.CM01.messagePrefix[0..2] := 'CM01 ';
   EM05.CM02.messagePrefix[0..2] := 'CM02 ';
   EM05.CM03.messagePrefix[0..2] := 'CM03 ';
   EM05.CM04.messagePrefix[0..2] := 'CM04 ';
   EM05.CM05.messagePrefix[0..2] := 'CM05 ';
   EM05.CM06.messagePrefix[0..2] := 'CM06 ';
   EM05.CM07.messagePrefix[0..2] := 'CM07 ';
   EM05.CM08.messagePrefix[0..2] := 'CM08 ';
   EM05.CM09.messagePrefix[0..2] := 'CM09 ';
   EM05.CM10.messagePrefix[0..2] := 'CM10 ';
   EM06.EventControl.messagePrefix[0..2] := 'EM06 ';
   EM06.CM01.messagePrefix[0..2] := 'CM01 ';
   EM06.CM02.messagePrefix[0..2] := 'CM02 ';
   EM06.CM03.messagePrefix[0..2] := 'CM03 ';
   EM06.CM04.messagePrefix[0..2] := 'CM04 ';
   EM06.CM05.messagePrefix[0..2] := 'CM05 ';
   EM06.CM06.messagePrefix[0..2] := 'CM06 ';
   EM06.CM07.messagePrefix[0..2] := 'CM07 ';
   EM06.CM08.messagePrefix[0..2] := 'CM08 ';
   EM06.CM09.messagePrefix[0..2] := 'CM09 ';
   EM06.CM10.messagePrefix[0..2] := 'CM10 ';
   EM07.EventControl.messagePrefix[0..2] := 'EM07 ';
   EM07.CM01.messagePrefix[0..2] := 'CM01 ';
   EM07.CM02.messagePrefix[0..2] := 'CM02 ';
   EM07.CM03.messagePrefix[0..2] := 'CM03 ';
   EM07.CM04.messagePrefix[0..2] := 'CM04 ';
   EM07.CM05.messagePrefix[0..2] := 'CM05 ';
   EM07.CM06.messagePrefix[0..2] := 'CM06 ';
   EM07.CM07.messagePrefix[0..2] := 'CM07 ';
   EM07.CM08.messagePrefix[0..2] := 'CM08 ';
   EM07.CM09.messagePrefix[0..2] := 'CM09 ';
   EM07.CM10.messagePrefix[0..2] := 'CM10 ';
   EM08.EventControl.messagePrefix[0..2] := 'EM08 ';
   EM08.CM01.messagePrefix[0..2] := 'CM01 ';
   EM08.CM02.messagePrefix[0..2] := 'CM02 ';
   EM08.CM03.messagePrefix[0..2] := 'CM03 ';
   EM08.CM04.messagePrefix[0..2] := 'CM04 ';
   EM08.CM05.messagePrefix[0..2] := 'CM05 ';
   EM08.CM06.messagePrefix[0..2] := 'CM06 ';
   EM08.CM07.messagePrefix[0..2] := 'CM07 ';
   EM08.CM08.messagePrefix[0..2] := 'CM08 ';
   EM08.CM09.messagePrefix[0..2] := 'CM09 ';
   EM08.CM10.messagePrefix[0..2] := 'CM10 ';
   EM09.EventControl.messagePrefix[0..2] := 'EM09 ';
   EM09.CM01.messagePrefix[0..2] := 'CM01 ';
   EM09.CM02.messagePrefix[0..2] := 'CM02 ';
   EM09.CM03.messagePrefix[0..2] := 'CM03 ';
   EM09.CM04.messagePrefix[0..2] := 'CM04 ';
   EM09.CM05.messagePrefix[0..2] := 'CM05 ';
   EM09.CM06.messagePrefix[0..2] := 'CM06 ';
   EM09.CM07.messagePrefix[0..2] := 'CM07 ';
   EM09.CM08.messagePrefix[0..2] := 'CM08 ';
   EM09.CM09.messagePrefix[0..2] := 'CM09 ';
   EM09.CM10.messagePrefix[0..2] := 'CM10 ';
END_DATA_BLOCK

